LIN {X 0,Y 488.725,Z 711.254,A -85,B 0,C 180,E1 -6470.898,E2 -6470.898} C_VEL
LIN {X 0,Y 488.408,Z 718.913,A -85,B 0,C 180,E1 -6472.143,E2 -6472.143} C_VEL
LIN {X 0,Y 488.185,Z 725.016,A -85,B 0,C 180,E1 -6473.386,E2 -6473.386} C_VEL
LIN {X 0,Y 488.072,Z 729.849,A -85,B 0,C 180,E1 -6474.629,E2 -6474.629} C_VEL
LIN {X 0,Y 488.106,Z 733.551,A -85,B 0,C 180,E1 -6475.871,E2 -6475.871} C_VEL
LIN {X 0,Y 487.981,Z 735.461,A -85,B 0,C 180,E1 -6476.697,E2 -6476.697} C_VEL
LIN {X 0,Y 487.99,Z 736.936,A -85,B 0,C 180,E1 -6477.524,E2 -6477.524} C_VEL
LIN {X 0,Y 487.835,Z 738.611,A -85,B 0,C 180,E1 -6479.174,E2 -6479.174} C_VEL
LIN {X 0,Y 487.82,Z 738.869,A -85,B 0,C 180,E1 -6480,E2 -6480} C_VEL
LIN {X 0,Y 487.835,Z 738.688,A -85,B 0,C 180,E1 -6480.825,E2 -6480.825} C_VEL
LIN {X 0,Y 487.989,Z 737.13,A -85,B 0,C 180,E1 -6482.476,E2 -6482.476} C_VEL
LIN {X 0,Y 487.981,Z 735.745,A -85,B 0,C 180,E1 -6483.302,E2 -6483.302} C_VEL
LIN {X 0,Y 488.067,Z 732.834,A -85,B 0,C 180,E1 -6484.542,E2 -6484.542} C_VEL
LIN {X 0,Y 488.225,Z 727.776,A -85,B 0,C 180,E1 -6486.069,E2 -6486.069} C_VEL
LIN {X 0,Y 488.344,Z 721.731,A -85,B 0,C 180,E1 -6487.442,E2 -6487.442} C_VEL
LIN {X 0,Y 488.606,Z 714.719,A -85,B 0,C 180,E1 -6488.687,E2 -6488.687} C_VEL
LIN {X 0,Y 488.878,Z 705.985,A -85,B 0,C 180,E1 -6489.934,E2 -6489.934} C_VEL
LIN {X 0,Y 489.234,Z 696.973,A -85,B 0,C 180,E1 -6490.973,E2 -6490.973} C_VEL
LIN {X 0,Y 489.603,Z 686.95,A -85,B 0,C 180,E1 -6491.908,E2 -6491.908} C_VEL
LIN {X 0,Y 489.945,Z 676.115,A -85,B 0,C 180,E1 -6492.727,E2 -6492.727} C_VEL
LIN {X 0,Y 490.19,Z 664.496,A -85,B 0,C 180,E1 -6493.42,E2 -6493.42} C_VEL
LIN {X 0,Y 490.575,Z 651.519,A -85,B 0,C 180,E1 -6493.99,E2 -6493.99} C_VEL
LIN {X 0,Y 490.841,Z 638.811,A -85,B 0,C 180,E1 -6494.379,E2 -6494.379} C_VEL
LIN {X 0,Y 491.087,Z 617.625,A -85,B 0,C 180,E1 -6494.742,E2 -6494.742} C_VEL
LIN {X 0,Y 491.674,Z 537.749,A -85,B 0,C 180,E1 -6496.029,E2 -6496.029} C_VEL
LIN {X 0,Y 489.935,Z 527.319,A -85,B 0,C 180,E1 -6496.278,E2 -6496.278} C_VEL
LIN {X 0,Y 490.381,Z 507.251,A -85,B 0,C 180,E1 -6499.246,E2 -6499.246} C_VEL
LIN {X 0,Y 490.847,Z 487.873,A -85,B 0,C 180,E1 -6502.077,E2 -6502.077} C_VEL
LIN {X 0,Y 490.974,Z 472.353,A -85,B 0,C 180,E1 -6504.301,E2 -6504.301} C_VEL
LIN {X 0,Y 488.784,Z 461.229,A -85,B 0,C 180,E1 -6506.011,E2 -6506.011} C_VEL
LIN {X 0,Y 488.728,Z 461.234,A -85,B 0,C 180,E1 -6509.27,E2 -6509.27} C_VEL
LIN {X 0,Y 488.708,Z 461.238,A -85,B 0,C 180,E1 -6512.147,E2 -6512.147} C_VEL
LIN {X 0,Y 488.728,Z 461.23,A -85,B 0,C 180,E1 -6515.114,E2 -6515.114} C_VEL
LIN {X 0,Y 488.685,Z 461.239,A -85,B 0,C 180,E1 -6518.2,E2 -6518.2} C_VEL
LIN {X 0,Y 488.723,Z 461.233,A -85,B 0,C 180,E1 -6520.344,E2 -6520.344} C_VEL
LIN {X 0,Y 488.688,Z 461.238,A -85,B 0,C 180,E1 -6523.654,E2 -6523.654} C_VEL
LIN {X 0,Y 488.689,Z 461.236,A -85,B 0,C 180,E1 -6526.345,E2 -6526.345} C_VEL
LIN {X 0,Y 488.737,Z 461.233,A -85,B 0,C 180,E1 -6529.676,E2 -6529.676} C_VEL
LIN {X 0,Y 488.683,Z 461.234,A -85,B 0,C 180,E1 -6532.841,E2 -6532.841} C_VEL
LIN {X 0,Y 488.735,Z 461.233,A -85,B 0,C 180,E1 -6535.887,E2 -6535.887} C_VEL
LIN {X 0,Y 488.696,Z 461.236,A -85,B 0,C 180,E1 -6538.82,E2 -6538.82} C_VEL
LIN {X 0,Y 488.771,Z 461.307,A -85,B 0,C 180,E1 -6542.154,E2 -6542.154} C_VEL
LIN {X 0,Y 492.591,Z 477.034,A -85,B 0,C 180,E1 -6544.507,E2 -6544.507} C_VEL
LIN {X 0,Y 492.585,Z 483.249,A -85,B 0,C 180,E1 -6545.333,E2 -6545.333} C_VEL
LIN {X 0,Y 491.403,Z 507.9,A -85,B 0,C 180,E1 -6548.515,E2 -6548.515} C_VEL
LIN {X 0,Y 490.794,Z 523.179,A -85,B 0,C 180,E1 -6550.474,E2 -6550.474} C_VEL
LIN {X 0,Y 493.097,Z 539.069,A -85,B 0,C 180,E1 -6550.81,E2 -6550.81} C_VEL
LIN {X 0,Y 491.916,Z 660.89,A -85,B 0,C 180,E1 -6552.701,E2 -6552.701} C_VEL
LIN {X 0,Y 491.605,Z 675.258,A -85,B 0,C 180,E1 -6553.091,E2 -6553.091} C_VEL
LIN {X 0,Y 491.241,Z 688.698,A -85,B 0,C 180,E1 -6553.617,E2 -6553.617} C_VEL
LIN {X 0,Y 490.769,Z 702.208,A -85,B 0,C 180,E1 -6554.317,E2 -6554.317} C_VEL
LIN {X 0,Y 490.228,Z 714.884,A -85,B 0,C 180,E1 -6555.151,E2 -6555.151} C_VEL
LIN {X 0,Y 489.715,Z 726.469,A -85,B 0,C 180,E1 -6556.09,E2 -6556.09} C_VEL
LIN {X 0,Y 489.278,Z 737.113,A -85,B 0,C 180,E1 -6557.135,E2 -6557.135} C_VEL
LIN {X 0,Y 488.939,Z 747.693,A -85,B 0,C 180,E1 -6558.39,E2 -6558.39} C_VEL
LIN {X 0,Y 488.572,Z 756.397,A -85,B 0,C 180,E1 -6559.64,E2 -6559.64} C_VEL
LIN {X 0,Y 488.293,Z 764.689,A -85,B 0,C 180,E1 -6561.098,E2 -6561.098} C_VEL
LIN {X 0,Y 488.084,Z 771.358,A -85,B 0,C 180,E1 -6562.553,E2 -6562.553} C_VEL
LIN {X 0,Y 488.006,Z 776.018,A -85,B 0,C 180,E1 -6563.81,E2 -6563.81} C_VEL
LIN {X 0,Y 487.962,Z 779.592,A -85,B 0,C 180,E1 -6565.041,E2 -6565.041} C_VEL
LIN {X 0,Y 487.959,Z 783.12,A -85,B 0,C 180,E1 -6566.696,E2 -6566.696} C_VEL
LIN {X 0,Y 487.985,Z 784.341,A -85,B 0,C 180,E1 -6567.523,E2 -6567.523} C_VEL
LIN {X 0,Y 487.831,Z 785.722,A -85,B 0,C 180,E1 -6569.173,E2 -6569.173} C_VEL
LIN {X 0,Y 487.83,Z 785.724,A -85,B 0,C 180,E1 -6570.824,E2 -6570.824} C_VEL
LIN {X 0,Y 487.985,Z 784.348,A -85,B 0,C 180,E1 -6572.475,E2 -6572.475} C_VEL
LIN {X 0,Y 487.935,Z 781.551,A -85,B 0,C 180,E1 -6574.129,E2 -6574.129} C_VEL
LIN {X 0,Y 488.022,Z 777.273,A -85,B 0,C 180,E1 -6575.784,E2 -6575.784} C_VEL
LIN {X 0,Y 488.082,Z 771.371,A -85,B 0,C 180,E1 -6577.445,E2 -6577.445} C_VEL
LIN {X 0,Y 488.288,Z 764.706,A -85,B 0,C 180,E1 -6578.9,E2 -6578.9} C_VEL
LIN {X 0,Y 488.577,Z 756.411,A -85,B 0,C 180,E1 -6580.357,E2 -6580.357} C_VEL
LIN {X 0,Y 488.942,Z 747.71,A -85,B 0,C 180,E1 -6581.608,E2 -6581.608} C_VEL
LIN {X 0,Y 489.302,Z 737.14,A -85,B 0,C 180,E1 -6582.862,E2 -6582.862} C_VEL
LIN {X 0,Y 489.779,Z 725.303,A -85,B 0,C 180,E1 -6584.012,E2 -6584.012} C_VEL
LIN {X 0,Y 490.304,Z 713.471,A -85,B 0,C 180,E1 -6584.951,E2 -6584.951} C_VEL
LIN {X 0,Y 490.815,Z 700.451,A -85,B 0,C 180,E1 -6585.786,E2 -6585.786} C_VEL
LIN {X 0,Y 491.313,Z 686.044,A -85,B 0,C 180,E1 -6586.503,E2 -6586.503} C_VEL
LIN {X 0,Y 491.653,Z 672.054,A -85,B 0,C 180,E1 -6587.012,E2 -6587.012} C_VEL
LIN {X 0,Y 491.999,Z 658.343,A -85,B 0,C 180,E1 -6587.348,E2 -6587.348} C_VEL
LIN {X 0,Y 493.037,Z 537.881,A -85,B 0,C 180,E1 -6589.211,E2 -6589.211} C_VEL
LIN {X 0,Y 490.784,Z 522.893,A -85,B 0,C 180,E1 -6589.547,E2 -6589.547} C_VEL
LIN {X 0,Y 491.888,Z 496.801,A -85,B 0,C 180,E1 -6592.912,E2 -6592.912} C_VEL
LIN {X 0,Y 492.731,Z 478.183,A -85,B 0,C 180,E1 -6595.333,E2 -6595.333} C_VEL
LIN {X 0,Y 489.178,Z 462.917,A -85,B 0,C 180,E1 -6597.601,E2 -6597.601} C_VEL
LIN {X 0,Y 488.747,Z 461.229,A -85,B 0,C 180,E1 -6597.86,E2 -6597.86} C_VEL
LIN {X 0,Y 488.715,Z 461.232,A -85,B 0,C 180,E1 -6600.364,E2 -6600.364} C_VEL
LIN {X 0,Y 488.731,Z 461.229,A -85,B 0,C 180,E1 -6603.483,E2 -6603.483} C_VEL
LIN {X 0,Y 488.684,Z 461.233,A -85,B 0,C 180,E1 -6606.355,E2 -6606.355} C_VEL
LIN {X 0,Y 488.743,Z 461.229,A -85,B 0,C 180,E1 -6609.248,E2 -6609.248} C_VEL
LIN {X 0,Y 488.727,Z 461.234,A -85,B 0,C 180,E1 -6612.52,E2 -6612.52} C_VEL
LIN {X 0,Y 488.704,Z 461.232,A -85,B 0,C 180,E1 -6615.198,E2 -6615.198} C_VEL
LIN {X 0,Y 488.727,Z 461.226,A -85,B 0,C 180,E1 -6617.478,E2 -6617.478} C_VEL
LIN {X 0,Y 488.74,Z 461.231,A -85,B 0,C 180,E1 -6620.75,E2 -6620.75} C_VEL
LIN {X 0,Y 488.676,Z 461.226,A -85,B 0,C 180,E1 -6623.868,E2 -6623.868} C_VEL
LIN {X 0,Y 488.73,Z 461.232,A -85,B 0,C 180,E1 -6626.877,E2 -6626.877} C_VEL
LIN {X 0,Y 488.724,Z 461.227,A -85,B 0,C 180,E1 -6629.781,E2 -6629.781} C_VEL
LIN {X 0,Y 488.788,Z 461.223,A -85,B 0,C 180,E1 -6633.054,E2 -6633.054} C_VEL
LIN {X 0,Y 488.683,Z 461.234,A -85,B 0,C 180,E1 -6636.254,E2 -6636.254} C_VEL
LIN {X 0,Y 488.735,Z 461.223,A -85,B 0,C 180,E1 -6639.175,E2 -6639.175} C_VEL
LIN {X 0,Y 488.748,Z 461.225,A -85,B 0,C 180,E1 -6641.627,E2 -6641.627} C_VEL
LIN {X 0,Y 488.75,Z 461.228,A -85,B 0,C 180,E1 -6644.999,E2 -6644.999} C_VEL
LIN {X 0,Y 488.822,Z 461.22,A -85,B 0,C 180,E1 -6648.388,E2 -6648.388} C_VEL
LIN {X 0,Y 488.807,Z 461.218,A -85,B 0,C 180,E1 -6651.734,E2 -6651.734} C_VEL
LIN {X 0,Y 488.852,Z 461.211,A -85,B 0,C 180,E1 -6654.224,E2 -6654.224} C_VEL
LIN {X 0,Y 488.952,Z 461.198,A -85,B 0,C 180,E1 -6657.529,E2 -6657.529} C_VEL
LIN {X 0,Y 488.958,Z 461.199,A -85,B 0,C 180,E1 -6660,E2 -6660} C_VEL
LIN {X 0,Y 488.951,Z 461.205,A -85,B 0,C 180,E1 -6662.472,E2 -6662.472} C_VEL
LIN {X 0,Y 488.845,Z 461.213,A -85,B 0,C 180,E1 -6665.776,E2 -6665.776} C_VEL
LIN {X 0,Y 488.808,Z 461.22,A -85,B 0,C 180,E1 -6668.267,E2 -6668.267} C_VEL
LIN {X 0,Y 488.819,Z 461.216,A -85,B 0,C 180,E1 -6671.612,E2 -6671.612} C_VEL
LIN {X 0,Y 488.754,Z 461.227,A -85,B 0,C 180,E1 -6675.001,E2 -6675.001} C_VEL
LIN {X 0,Y 488.744,Z 461.229,A -85,B 0,C 180,E1 -6678.443,E2 -6678.443} C_VEL
LIN {X 0,Y 488.697,Z 461.232,A -85,B 0,C 180,E1 -6681.071,E2 -6681.071} C_VEL
LIN {X 0,Y 488.684,Z 461.233,A -85,B 0,C 180,E1 -6683.746,E2 -6683.746} C_VEL
LIN {X 0,Y 488.789,Z 461.222,A -85,B 0,C 180,E1 -6686.946,E2 -6686.946} C_VEL
LIN {X 0,Y 488.71,Z 461.234,A -85,B 0,C 180,E1 -6690.366,E2 -6690.366} C_VEL
LIN {X 0,Y 488.728,Z 461.226,A -85,B 0,C 180,E1 -6693.486,E2 -6693.486} C_VEL
LIN {X 0,Y 488.682,Z 461.241,A -85,B 0,C 180,E1 -6696.357,E2 -6696.357} C_VEL
LIN {X 0,Y 488.741,Z 461.227,A -85,B 0,C 180,E1 -6699.251,E2 -6699.251} C_VEL
LIN {X 0,Y 488.684,Z 461.24,A -85,B 0,C 180,E1 -6702.527,E2 -6702.527} C_VEL
LIN {X 0,Y 488.706,Z 461.231,A -85,B 0,C 180,E1 -6705.2,E2 -6705.2} C_VEL
LIN {X 0,Y 488.73,Z 461.228,A -85,B 0,C 180,E1 -6707.481,E2 -6707.481} C_VEL
LIN {X 0,Y 488.745,Z 461.231,A -85,B 0,C 180,E1 -6710.752,E2 -6710.752} C_VEL
LIN {X 0,Y 488.682,Z 461.233,A -85,B 0,C 180,E1 -6713.87,E2 -6713.87} C_VEL
LIN {X 0,Y 488.736,Z 461.232,A -85,B 0,C 180,E1 -6716.879,E2 -6716.879} C_VEL
LIN {X 0,Y 488.732,Z 461.231,A -85,B 0,C 180,E1 -6719.783,E2 -6719.783} C_VEL
LIN {X 0,Y 488.792,Z 461.226,A -85,B 0,C 180,E1 -6723.11,E2 -6723.11} C_VEL
LIN {X 0,Y 488.533,Z 461.627,A -85,B 0,C 180,E1 -6723.564,E2 -6723.564} C_VEL
LIN {X 0,Y 487.572,Z 463.402,A -85,B 0,C 180,E1 -6724.212,E2 -6724.212} C_VEL
LIN {X 0,Y 486.316,Z 466.116,A -85,B 0,C 180,E1 -6724.816,E2 -6724.816} C_VEL
LIN {X 0,Y 484.792,Z 470.694,A -85,B 0,C 180,E1 -6725.6,E2 -6725.6} C_VEL
LIN {X 0,Y 484.379,Z 475.251,A -85,B 0,C 180,E1 -6726.389,E2 -6726.389} C_VEL
LIN {X 0,Y 483.995,Z 487.151,A -85,B 0,C 180,E1 -6728.472,E2 -6728.472} C_VEL
LIN {X 0,Y 483.111,Z 507.748,A -85,B 0,C 180,E1 -6731.994,E2 -6731.994} C_VEL
LIN {X 0,Y 482.787,Z 515.697,A -85,B 0,C 180,E1 -6733.327,E2 -6733.327} C_VEL
LIN {X 0,Y 485.47,Z 530.483,A -85,B 0,C 180,E1 -6733.646,E2 -6733.646} C_VEL
LIN {X 0,Y 485.028,Z 626.011,A -85,B 0,C 180,E1 -6734.99,E2 -6734.99} C_VEL
LIN {X 0,Y 484.776,Z 638.769,A -85,B 0,C 180,E1 -6735.331,E2 -6735.331} C_VEL
LIN {X 0,Y 484.401,Z 651.155,A -85,B 0,C 180,E1 -6735.829,E2 -6735.829} C_VEL
LIN {X 0,Y 484.02,Z 662.666,A -85,B 0,C 180,E1 -6736.461,E2 -6736.461} C_VEL
LIN {X 0,Y 483.555,Z 673.193,A -85,B 0,C 180,E1 -6737.201,E2 -6737.201} C_VEL
LIN {X 0,Y 483.049,Z 683.796,A -85,B 0,C 180,E1 -6738.142,E2 -6738.142} C_VEL
LIN {X 0,Y 482.618,Z 692.492,A -85,B 0,C 180,E1 -6739.089,E2 -6739.089} C_VEL
LIN {X 0,Y 482.109,Z 701.921,A -85,B 0,C 180,E1 -6740.35,E2 -6740.35} C_VEL
LIN {X 0,Y 481.674,Z 709.481,A -85,B 0,C 180,E1 -6741.611,E2 -6741.611} C_VEL
LIN {X 0,Y 481.359,Z 715.713,A -85,B 0,C 180,E1 -6742.914,E2 -6742.914} C_VEL
LIN {X 0,Y 481.15,Z 720.373,A -85,B 0,C 180,E1 -6744.133,E2 -6744.133} C_VEL
LIN {X 0,Y 481.041,Z 724.131,A -85,B 0,C 180,E1 -6745.392,E2 -6745.392} C_VEL
LIN {X 0,Y 480.984,Z 726.915,A -85,B 0,C 180,E1 -6746.65,E2 -6746.65} C_VEL
LIN {X 0,Y 480.939,Z 728.241,A -85,B 0,C 180,E1 -6747.489,E2 -6747.489} C_VEL
LIN {X 0,Y 480.762,Z 729.781,A -85,B 0,C 180,E1 -6749.163,E2 -6749.163} C_VEL
LIN {X 0,Y 480.748,Z 730.004,A -85,B 0,C 180,E1 -6750.001,E2 -6750.001} C_VEL
LIN {X 0,Y 480.826,Z 729.271,A -85,B 0,C 180,E1 -6751.676,E2 -6751.676} C_VEL
LIN {X 0,Y 480.937,Z 728.348,A -85,B 0,C 180,E1 -6752.514,E2 -6752.514} C_VEL
LIN {X 0,Y 480.961,Z 727.06,A -85,B 0,C 180,E1 -6753.352,E2 -6753.352} C_VEL
LIN {X 0,Y 481.034,Z 724.342,A -85,B 0,C 180,E1 -6754.61,E2 -6754.61} C_VEL
LIN {X 0,Y 481.147,Z 720.657,A -85,B 0,C 180,E1 -6755.87,E2 -6755.87} C_VEL
LIN {X 0,Y 481.397,Z 715.111,A -85,B 0,C 180,E1 -6757.319,E2 -6757.319} C_VEL
LIN {X 0,Y 481.726,Z 708.806,A -85,B 0,C 180,E1 -6758.601,E2 -6758.601} C_VEL
LIN {X 0,Y 482.108,Z 701.082,A -85,B 0,C 180,E1 -6759.864,E2 -6759.864} C_VEL
LIN {X 0,Y 482.615,Z 691.481,A -85,B 0,C 180,E1 -6761.126,E2 -6761.126} C_VEL
LIN {X 0,Y 483.177,Z 681.429,A -85,B 0,C 180,E1 -6762.177,E2 -6762.177} C_VEL
LIN {X 0,Y 483.684,Z 670.239,A -85,B 0,C 180,E1 -6763.111,E2 -6763.111} C_VEL
LIN {X 0,Y 484.171,Z 658.857,A -85,B 0,C 180,E1 -6763.858,E2 -6763.858} C_VEL
LIN {X 0,Y 484.577,Z 647.318,A -85,B 0,C 180,E1 -6764.436,E2 -6764.436} C_VEL
LIN {X 0,Y 484.864,Z 634.808,A -85,B 0,C 180,E1 -6764.883,E2 -6764.883} C_VEL
LIN {X 0,Y 485.089,Z 621.87,A -85,B 0,C 180,E1 -6765.171,E2 -6765.171} C_VEL
LIN {X 0,Y 485.331,Z 529.087,A -85,B 0,C 180,E1 -6766.469,E2 -6766.469} C_VEL
LIN {X 0,Y 482.801,Z 515.558,A -85,B 0,C 180,E1 -6766.786,E2 -6766.786} C_VEL
LIN {X 0,Y 483.399,Z 499.245,A -85,B 0,C 180,E1 -6769.536,E2 -6769.536} C_VEL
LIN {X 0,Y 484.17,Z 482.676,A -85,B 0,C 180,E1 -6772.399,E2 -6772.399} C_VEL
LIN {X 0,Y 484.393,Z 475.065,A -85,B 0,C 180,E1 -6773.734,E2 -6773.734} C_VEL
LIN {X 0,Y 481.723,Z 462.108,A -85,B 0,C 180,E1 -6776.248,E2 -6776.248} C_VEL
LIN {X 0,Y 481.684,Z 462.113,A -85,B 0,C 180,E1 -6778.904,E2 -6778.904} C_VEL
LIN {X 0,Y 481.663,Z 462.113,A -85,B 0,C 180,E1 -6782.19,E2 -6782.19} C_VEL
LIN {X 0,Y 481.694,Z 462.105,A -85,B 0,C 180,E1 -6784.683,E2 -6784.683} C_VEL
LIN {X 0,Y 481.661,Z 462.111,A -85,B 0,C 180,E1 -6788.008,E2 -6788.008} C_VEL
LIN {X 0,Y 481.669,Z 462.108,A -85,B 0,C 180,E1 -6791.041,E2 -6791.041} C_VEL
LIN {X 0,Y 481.665,Z 462.106,A -85,B 0,C 180,E1 -6794.36,E2 -6794.36} C_VEL
LIN {X 0,Y 481.649,Z 462.11,A -85,B 0,C 180,E1 -6796.852,E2 -6796.852} C_VEL
LIN {X 0,Y 481.683,Z 462.108,A -85,B 0,C 180,E1 -6800.06,E2 -6800.06} C_VEL
LIN {X 0,Y 481.635,Z 462.111,A -85,B 0,C 180,E1 -6803.254,E2 -6803.254} C_VEL
LIN {X 0,Y 481.716,Z 462.103,A -85,B 0,C 180,E1 -6806.33,E2 -6806.33} C_VEL
LIN {X 0,Y 481.657,Z 462.114,A -85,B 0,C 180,E1 -6809.417,E2 -6809.417} C_VEL
LIN {X 0,Y 481.706,Z 462.107,A -85,B 0,C 180,E1 -6812.168,E2 -6812.168} C_VEL
LIN {X 0,Y 481.761,Z 462.29,A -85,B 0,C 180,E1 -6813.61,E2 -6813.61} C_VEL
LIN {X 0,Y 484.205,Z 474.142,A -85,B 0,C 180,E1 -6815.565,E2 -6815.565} C_VEL
LIN {X 0,Y 484.167,Z 483.006,A -85,B 0,C 180,E1 -6816.926,E2 -6816.926} C_VEL
LIN {X 0,Y 483.541,Z 503.362,A -85,B 0,C 180,E1 -6820.028,E2 -6820.028} C_VEL
LIN {X 0,Y 482.967,Z 523.364,A -85,B 0,C 180,E1 -6823.08,E2 -6823.08} C_VEL
LIN {X 0,Y 482.888,Z 526.537,A -85,B 0,C 180,E1 -6823.562,E2 -6823.562} C_VEL
LIN {X 0,Y 484.92,Z 539.144,A -85,B 0,C 180,E1 -6823.859,E2 -6823.859} C_VEL
LIN {X 0,Y 483.987,Z 636.668,A -85,B 0,C 180,E1 -6825.44,E2 -6825.44} C_VEL
LIN {X 0,Y 483.758,Z 649.432,A -85,B 0,C 180,E1 -6825.809,E2 -6825.809} C_VEL
LIN {X 0,Y 483.415,Z 661.772,A -85,B 0,C 180,E1 -6826.335,E2 -6826.335} C_VEL
LIN {X 0,Y 483.085,Z 673.368,A -85,B 0,C 180,E1 -6826.993,E2 -6826.993} C_VEL
LIN {X 0,Y 482.756,Z 684.635,A -85,B 0,C 180,E1 -6827.813,E2 -6827.813} C_VEL
LIN {X 0,Y 482.283,Z 696.06,A -85,B 0,C 180,E1 -6828.867,E2 -6828.867} C_VEL
LIN {X 0,Y 481.923,Z 705.281,A -85,B 0,C 180,E1 -6829.921,E2 -6829.921} C_VEL
LIN {X 0,Y 481.586,Z 714.167,A -85,B 0,C 180,E1 -6831.186,E2 -6831.186} C_VEL
LIN {X 0,Y 481.289,Z 721.327,A -85,B 0,C 180,E1 -6832.448,E2 -6832.448} C_VEL
LIN {X 0,Y 481.135,Z 726.739,A -85,B 0,C 180,E1 -6833.637,E2 -6833.637} C_VEL
LIN {X 0,Y 480.915,Z 731.506,A -85,B 0,C 180,E1 -6834.97,E2 -6834.97} C_VEL
LIN {X 0,Y 481.021,Z 733.841,A -85,B 0,C 180,E1 -6835.811,E2 -6835.811} C_VEL
LIN {X 0,Y 480.913,Z 735.764,A -85,B 0,C 180,E1 -6836.649,E2 -6836.649} C_VEL
LIN {X 0,Y 480.897,Z 737.251,A -85,B 0,C 180,E1 -6837.487,E2 -6837.487} C_VEL
LIN {X 0,Y 480.761,Z 738.938,A -85,B 0,C 180,E1 -6839.162,E2 -6839.162} C_VEL
LIN {X 0,Y 480.744,Z 739.2,A -85,B 0,C 180,E1 -6840,E2 -6840} C_VEL
LIN {X 0,Y 480.761,Z 739.019,A -85,B 0,C 180,E1 -6840.837,E2 -6840.837} C_VEL
LIN {X 0,Y 480.911,Z 737.457,A -85,B 0,C 180,E1 -6842.513,E2 -6842.513} C_VEL
LIN {X 0,Y 480.913,Z 736.064,A -85,B 0,C 180,E1 -6843.351,E2 -6843.351} C_VEL
LIN {X 0,Y 480.982,Z 733.14,A -85,B 0,C 180,E1 -6844.609,E2 -6844.609} C_VEL
LIN {X 0,Y 481.134,Z 729.148,A -85,B 0,C 180,E1 -6845.869,E2 -6845.869} C_VEL
LIN {X 0,Y 481.209,Z 723.972,A -85,B 0,C 180,E1 -6847.131,E2 -6847.131} C_VEL
LIN {X 0,Y 481.49,Z 717.445,A -85,B 0,C 180,E1 -6848.393,E2 -6848.393} C_VEL
LIN {X 0,Y 481.738,Z 709.334,A -85,B 0,C 180,E1 -6849.658,E2 -6849.658} C_VEL
LIN {X 0,Y 482.079,Z 700.952,A -85,B 0,C 180,E1 -6850.712,E2 -6850.712} C_VEL
LIN {X 0,Y 482.522,Z 690.632,A -85,B 0,C 180,E1 -6851.766,E2 -6851.766} C_VEL
LIN {X 0,Y 482.886,Z 680.426,A -85,B 0,C 180,E1 -6852.61,E2 -6852.61} C_VEL
LIN {X 0,Y 483.182,Z 668.326,A -85,B 0,C 180,E1 -6853.399,E2 -6853.399} C_VEL
LIN {X 0,Y 483.583,Z 655.358,A -85,B 0,C 180,E1 -6854.035,E2 -6854.035} C_VEL
LIN {X 0,Y 483.889,Z 642.229,A -85,B 0,C 180,E1 -6854.482,E2 -6854.482} C_VEL
LIN {X 0,Y 484.068,Z 628.396,A -85,B 0,C 180,E1 -6854.773,E2 -6854.773} C_VEL
LIN {X 0,Y 484.879,Z 538.539,A -85,B 0,C 180,E1 -6856.253,E2 -6856.253} C_VEL
LIN {X 0,Y 483.066,Z 527.717,A -85,B 0,C 180,E1 -6856.527,E2 -6856.527} C_VEL
LIN {X 0,Y 483.499,Z 507.474,A -85,B 0,C 180,E1 -6859.531,E2 -6859.531} C_VEL
LIN {X 0,Y 483.941,Z 490.703,A -85,B 0,C 180,E1 -6862.003,E2 -6862.003} C_VEL
LIN {X 0,Y 484.299,Z 475.446,A -85,B 0,C 180,E1 -6864.202,E2 -6864.202} C_VEL
LIN {X 0,Y 482.705,Z 466.129,A -85,B 0,C 180,E1 -6865.626,E2 -6865.626} C_VEL
LIN {X 0,Y 481.73,Z 462.107,A -85,B 0,C 180,E1 -6866.275,E2 -6866.275} C_VEL
LIN {X 0,Y 481.683,Z 462.112,A -85,B 0,C 180,E1 -6868.903,E2 -6868.903} C_VEL
LIN {X 0,Y 481.662,Z 462.116,A -85,B 0,C 180,E1 -6872.189,E2 -6872.189} C_VEL
LIN {X 0,Y 481.698,Z 462.108,A -85,B 0,C 180,E1 -6874.681,E2 -6874.681} C_VEL
LIN {X 0,Y 481.66,Z 462.116,A -85,B 0,C 180,E1 -6878.007,E2 -6878.007} C_VEL
LIN {X 0,Y 481.661,Z 462.11,A -85,B 0,C 180,E1 -6881.041,E2 -6881.041} C_VEL
LIN {X 0,Y 481.659,Z 462.112,A -85,B 0,C 180,E1 -6884.457,E2 -6884.457} C_VEL
LIN {X 0,Y 481.652,Z 462.116,A -85,B 0,C 180,E1 -6887.839,E2 -6887.839} C_VEL
LIN {X 0,Y 481.665,Z 462.107,A -85,B 0,C 180,E1 -6890.653,E2 -6890.653} C_VEL
LIN {X 0,Y 481.632,Z 462.118,A -85,B 0,C 180,E1 -6893.376,E2 -6893.376} C_VEL
LIN {X 0,Y 481.714,Z 462.105,A -85,B 0,C 180,E1 -6896.329,E2 -6896.329} C_VEL
LIN {X 0,Y 481.655,Z 462.117,A -85,B 0,C 180,E1 -6899.417,E2 -6899.417} C_VEL
LIN {X 0,Y 481.709,Z 462.126,A -85,B 0,C 180,E1 -6901.842,E2 -6901.842} C_VEL
LIN {X 0,Y 485.587,Z 477.99,A -85,B 0,C 180,E1 -6904.265,E2 -6904.265} C_VEL
LIN {X 0,Y 485.926,Z 481.392,A -85,B 0,C 180,E1 -6904.743,E2 -6904.743} C_VEL
LIN {X 0,Y 484.664,Z 505.062,A -85,B 0,C 180,E1 -6907.85,E2 -6907.85} C_VEL
LIN {X 0,Y 483.87,Z 522.955,A -85,B 0,C 180,E1 -6910.197,E2 -6910.197} C_VEL
LIN {X 0,Y 486.32,Z 539.434,A -85,B 0,C 180,E1 -6910.563,E2 -6910.563} C_VEL
LIN {X 0,Y 485.078,Z 660.109,A -85,B 0,C 180,E1 -6912.476,E2 -6912.476} C_VEL
LIN {X 0,Y 484.722,Z 674.54,A -85,B 0,C 180,E1 -6912.871,E2 -6912.871} C_VEL
LIN {X 0,Y 484.35,Z 688.164,A -85,B 0,C 180,E1 -6913.41,E2 -6913.41} C_VEL
LIN {X 0,Y 483.851,Z 701.149,A -85,B 0,C 180,E1 -6914.087,E2 -6914.087} C_VEL
LIN {X 0,Y 483.294,Z 713.953,A -85,B 0,C 180,E1 -6914.933,E2 -6914.933} C_VEL
LIN {X 0,Y 482.774,Z 725.639,A -85,B 0,C 180,E1 -6915.886,E2 -6915.886} C_VEL
LIN {X 0,Y 482.279,Z 736.362,A -85,B 0,C 180,E1 -6916.945,E2 -6916.945} C_VEL
LIN {X 0,Y 481.917,Z 747.023,A -85,B 0,C 180,E1 -6918.218,E2 -6918.218} C_VEL
LIN {X 0,Y 481.529,Z 755.788,A -85,B 0,C 180,E1 -6919.487,E2 -6919.487} C_VEL
LIN {X 0,Y 481.225,Z 764.136,A -85,B 0,C 180,E1 -6920.966,E2 -6920.966} C_VEL
LIN {X 0,Y 481.009,Z 770.847,A -85,B 0,C 180,E1 -6922.443,E2 -6922.443} C_VEL
LIN {X 0,Y 480.909,Z 775.917,A -85,B 0,C 180,E1 -6923.841,E2 -6923.841} C_VEL
LIN {X 0,Y 480.896,Z 779.136,A -85,B 0,C 180,E1 -6924.968,E2 -6924.968} C_VEL
LIN {X 0,Y 480.884,Z 782.69,A -85,B 0,C 180,E1 -6926.648,E2 -6926.648} C_VEL
LIN {X 0,Y 480.822,Z 784.791,A -85,B 0,C 180,E1 -6928.324,E2 -6928.324} C_VEL
LIN {X 0,Y 480.741,Z 785.487,A -85,B 0,C 180,E1 -6929.999,E2 -6929.999} C_VEL
LIN {X 0,Y 480.822,Z 784.795,A -85,B 0,C 180,E1 -6931.674,E2 -6931.674} C_VEL
LIN {X 0,Y 480.883,Z 782.7,A -85,B 0,C 180,E1 -6933.35,E2 -6933.35} C_VEL
LIN {X 0,Y 480.896,Z 779.152,A -85,B 0,C 180,E1 -6935.029,E2 -6935.029} C_VEL
LIN {X 0,Y 480.961,Z 774.047,A -85,B 0,C 180,E1 -6936.712,E2 -6936.712} C_VEL
LIN {X 0,Y 481.08,Z 769.096,A -85,B 0,C 180,E1 -6937.976,E2 -6937.976} C_VEL
LIN {X 0,Y 481.332,Z 761.936,A -85,B 0,C 180,E1 -6939.453,E2 -6939.453} C_VEL
LIN {X 0,Y 481.657,Z 753.03,A -85,B 0,C 180,E1 -6940.933,E2 -6940.933} C_VEL
LIN {X 0,Y 481.908,Z 744.117,A -85,B 0,C 180,E1 -6942.153,E2 -6942.153} C_VEL
LIN {X 0,Y 482.459,Z 733.391,A -85,B 0,C 180,E1 -6943.37,E2 -6943.37} C_VEL
LIN {X 0,Y 482.962,Z 722.068,A -85,B 0,C 180,E1 -6944.429,E2 -6944.429} C_VEL
LIN {X 0,Y 483.529,Z 709.56,A -85,B 0,C 180,E1 -6945.381,E2 -6945.381} C_VEL
LIN {X 0,Y 483.983,Z 696.444,A -85,B 0,C 180,E1 -6946.18,E2 -6946.18} C_VEL
LIN {X 0,Y 484.433,Z 683.35,A -85,B 0,C 180,E1 -6946.801,E2 -6946.801} C_VEL
LIN {X 0,Y 484.864,Z 669.495,A -85,B 0,C 180,E1 -6947.285,E2 -6947.285} C_VEL
LIN {X 0,Y 485.2,Z 654.571,A -85,B 0,C 180,E1 -6947.626,E2 -6947.626} C_VEL
LIN {X 0,Y 486.307,Z 539.649,A -85,B 0,C 180,E1 -6949.432,E2 -6949.432} C_VEL
LIN {X 0,Y 483.91,Z 522.826,A -85,B 0,C 180,E1 -6949.813,E2 -6949.813} C_VEL
LIN {X 0,Y 485.006,Z 498.304,A -85,B 0,C 180,E1 -6953.031,E2 -6953.031} C_VEL
LIN {X 0,Y 485.887,Z 479.709,A -85,B 0,C 180,E1 -6955.486,E2 -6955.486} C_VEL
LIN {X 0,Y 482.247,Z 464.453,A -85,B 0,C 180,E1 -6957.796,E2 -6957.796} C_VEL
LIN {X 0,Y 481.716,Z 462.105,A -85,B 0,C 180,E1 -6958.184,E2 -6958.184} C_VEL
LIN {X 0,Y 481.649,Z 462.114,A -85,B 0,C 180,E1 -6960.709,E2 -6960.709} C_VEL
LIN {X 0,Y 481.691,Z 462.105,A -85,B 0,C 180,E1 -6963.732,E2 -6963.732} C_VEL
LIN {X 0,Y 481.625,Z 462.118,A -85,B 0,C 180,E1 -6966.745,E2 -6966.745} C_VEL
LIN {X 0,Y 481.687,Z 462.107,A -85,B 0,C 180,E1 -6969.938,E2 -6969.938} C_VEL
LIN {X 0,Y 481.677,Z 462.108,A -85,B 0,C 180,E1 -6973.294,E2 -6973.294} C_VEL
LIN {X 0,Y 481.681,Z 462.11,A -85,B 0,C 180,E1 -6976.845,E2 -6976.845} C_VEL
LIN {X 0,Y 481.684,Z 462.104,A -85,B 0,C 180,E1 -6980.06,E2 -6980.06} C_VEL
LIN {X 0,Y 481.621,Z 462.105,A -85,B 0,C 180,E1 -6983.253,E2 -6983.253} C_VEL
LIN {X 0,Y 481.699,Z 462.103,A -85,B 0,C 180,E1 -6986.329,E2 -6986.329} C_VEL
LIN {X 0,Y 481.649,Z 462.109,A -85,B 0,C 180,E1 -6989.415,E2 -6989.415} C_VEL
LIN {X 0,Y 481.692,Z 462.105,A -85,B 0,C 180,E1 -6992.168,E2 -6992.168} C_VEL
LIN {X 0,Y 481.708,Z 462.104,A -85,B 0,C 180,E1 -6994.969,E2 -6994.969} C_VEL
LIN {X 0,Y 481.642,Z 462.097,A -85,B 0,C 180,E1 -6997.704,E2 -6997.704} C_VEL
LIN {X 0,Y 481.697,Z 462.103,A -85,B 0,C 180,E1 -7000.393,E2 -7000.393} C_VEL
LIN {X 0,Y 481.681,Z 462.106,A -85,B 0,C 180,E1 -7003.034,E2 -7003.034} C_VEL
LIN {X 0,Y 481.68,Z 462.105,A -85,B 0,C 180,E1 -7005.639,E2 -7005.639} C_VEL
LIN {X 0,Y 481.784,Z 462.095,A -85,B 0,C 180,E1 -7008.216,E2 -7008.216} C_VEL
LIN {X 0,Y 481.753,Z 462.096,A -85,B 0,C 180,E1 -7011.612,E2 -7011.612} C_VEL
LIN {X 0,Y 481.812,Z 462.086,A -85,B 0,C 180,E1 -7014.14,E2 -7014.14} C_VEL
LIN {X 0,Y 481.919,Z 462.074,A -85,B 0,C 180,E1 -7017.493,E2 -7017.493} C_VEL
LIN {X 0,Y 481.929,Z 462.074,A -85,B 0,C 180,E1 -7020,E2 -7020} C_VEL
LIN {X 0,Y 481.918,Z 462.08,A -85,B 0,C 180,E1 -7022.508,E2 -7022.508} C_VEL
LIN {X 0,Y 481.806,Z 462.091,A -85,B 0,C 180,E1 -7025.861,E2 -7025.861} C_VEL
LIN {X 0,Y 481.753,Z 462.099,A -85,B 0,C 180,E1 -7028.389,E2 -7028.389} C_VEL
LIN {X 0,Y 481.784,Z 462.093,A -85,B 0,C 180,E1 -7031.784,E2 -7031.784} C_VEL
LIN {X 0,Y 481.733,Z 462.1,A -85,B 0,C 180,E1 -7035.225,E2 -7035.225} C_VEL
LIN {X 0,Y 481.702,Z 462.109,A -85,B 0,C 180,E1 -7038.722,E2 -7038.722} C_VEL
LIN {X 0,Y 481.637,Z 462.109,A -85,B 0,C 180,E1 -7041.395,E2 -7041.395} C_VEL
LIN {X 0,Y 481.667,Z 462.11,A -85,B 0,C 180,E1 -7044.114,E2 -7044.114} C_VEL
LIN {X 0,Y 481.742,Z 462.098,A -85,B 0,C 180,E1 -7047.141,E2 -7047.141} C_VEL
LIN {X 0,Y 481.679,Z 462.105,A -85,B 0,C 180,E1 -7049.741,E2 -7049.741} C_VEL
LIN {X 0,Y 481.665,Z 462.112,A -85,B 0,C 180,E1 -7052.675,E2 -7052.675} C_VEL
LIN {X 0,Y 481.636,Z 462.112,A -85,B 0,C 180,E1 -7055.71,E2 -7055.71} C_VEL
LIN {X 0,Y 481.712,Z 462.102,A -85,B 0,C 180,E1 -7059.356,E2 -7059.356} C_VEL
LIN {X 0,Y 481.642,Z 462.116,A -85,B 0,C 180,E1 -7062.162,E2 -7062.162} C_VEL
LIN {X 0,Y 481.654,Z 462.109,A -85,B 0,C 180,E1 -7065.544,E2 -7065.544} C_VEL
LIN {X 0,Y 481.668,Z 462.112,A -85,B 0,C 180,E1 -7068.086,E2 -7068.086} C_VEL
LIN {X 0,Y 481.699,Z 462.105,A -85,B 0,C 180,E1 -7071.145,E2 -7071.145} C_VEL
LIN {X 0,Y 481.665,Z 462.112,A -85,B 0,C 180,E1 -7074.796,E2 -7074.796} C_VEL
LIN {X 0,Y 481.671,Z 462.109,A -85,B 0,C 180,E1 -7077.327,E2 -7077.327} C_VEL
LIN {X 0,Y 481.686,Z 462.111,A -85,B 0,C 180,E1 -7080.261,E2 -7080.261} C_VEL
LIN {X 0,Y 481.726,Z 462.106,A -85,B 0,C 180,E1 -7083.58,E2 -7083.58} C_VEL
LIN {X 0,Y 481.754,Z 462.261,A -85,B 0,C 180,E1 -7083.902,E2 -7083.902} C_VEL
LIN {X 0,Y 484.379,Z 475.251,A -85,B 0,C 180,E1 -7086.389,E2 -7086.389} C_VEL
LIN {X 0,Y 483.925,Z 478.596,A -85,B 0,C 180,E1 -7086.958,E2 -7086.958} C_VEL
LIN {X 0,Y 482.338,Z 482.1,A -85,B 0,C 180,E1 -7087.494,E2 -7087.494} C_VEL
LIN {X 0,Y 477.7,Z 490.388,A -85,B 0,C 180,E1 -7088.725,E2 -7088.725} C_VEL
LIN {X 0,Y 476.799,Z 493.87,A -85,B 0,C 180,E1 -7089.297,E2 -7089.297} C_VEL
LIN {X 0,Y 476.06,Z 510.529,A -85,B 0,C 180,E1 -7092.163,E2 -7092.163} C_VEL
LIN {X 0,Y 475.886,Z 515.871,A -85,B 0,C 180,E1 -7093.056,E2 -7093.056} C_VEL
LIN {X 0,Y 478.725,Z 530.777,A -85,B 0,C 180,E1 -7093.387,E2 -7093.387} C_VEL
LIN {X 0,Y 478.249,Z 626.376,A -85,B 0,C 180,E1 -7094.745,E2 -7094.745} C_VEL
LIN {X 0,Y 477.989,Z 639.149,A -85,B 0,C 180,E1 -7095.091,E2 -7095.091} C_VEL
LIN {X 0,Y 477.578,Z 652.109,A -85,B 0,C 180,E1 -7095.622,E2 -7095.622} C_VEL
LIN {X 0,Y 477.17,Z 663.496,A -85,B 0,C 180,E1 -7096.262,E2 -7096.262} C_VEL
LIN {X 0,Y 476.67,Z 675.158,A -85,B 0,C 180,E1 -7097.119,E2 -7097.119} C_VEL
LIN {X 0,Y 476.022,Z 685.515,A -85,B 0,C 180,E1 -7098.072,E2 -7098.072} C_VEL
LIN {X 0,Y 475.569,Z 694.858,A -85,B 0,C 180,E1 -7099.141,E2 -7099.141} C_VEL
LIN {X 0,Y 475.157,Z 702.513,A -85,B 0,C 180,E1 -7100.208,E2 -7100.208} C_VEL
LIN {X 0,Y 474.69,Z 710.027,A -85,B 0,C 180,E1 -7101.487,E2 -7101.487} C_VEL
LIN {X 0,Y 474.328,Z 716.227,A -85,B 0,C 180,E1 -7102.809,E2 -7102.809} C_VEL
LIN {X 0,Y 474.109,Z 720.855,A -85,B 0,C 180,E1 -7104.045,E2 -7104.045} C_VEL
LIN {X 0,Y 473.982,Z 724.587,A -85,B 0,C 180,E1 -7105.323,E2 -7105.323} C_VEL
LIN {X 0,Y 473.912,Z 727.351,A -85,B 0,C 180,E1 -7106.6,E2 -7106.6} C_VEL
LIN {X 0,Y 473.88,Z 728.663,A -85,B 0,C 180,E1 -7107.451,E2 -7107.451} C_VEL
LIN {X 0,Y 473.691,Z 730.192,A -85,B 0,C 180,E1 -7109.151,E2 -7109.151} C_VEL
LIN {X 0,Y 473.674,Z 730.412,A -85,B 0,C 180,E1 -7110.001,E2 -7110.001} C_VEL
LIN {X 0,Y 473.761,Z 729.687,A -85,B 0,C 180,E1 -7111.701,E2 -7111.701} C_VEL
LIN {X 0,Y 473.878,Z 728.771,A -85,B 0,C 180,E1 -7112.551,E2 -7112.551} C_VEL
LIN {X 0,Y 473.995,Z 725.811,A -85,B 0,C 180,E1 -7114.253,E2 -7114.253} C_VEL
LIN {X 0,Y 473.981,Z 722.499,A -85,B 0,C 180,E1 -7115.532,E2 -7115.532} C_VEL
LIN {X 0,Y 474.243,Z 718.065,A -85,B 0,C 180,E1 -7116.829,E2 -7116.829} C_VEL
LIN {X 0,Y 474.587,Z 711.548,A -85,B 0,C 180,E1 -7118.303,E2 -7118.303} C_VEL
LIN {X 0,Y 475.004,Z 704.41,A -85,B 0,C 180,E1 -7119.583,E2 -7119.583} C_VEL
LIN {X 0,Y 475.515,Z 695.557,A -85,B 0,C 180,E1 -7120.863,E2 -7120.863} C_VEL
LIN {X 0,Y 475.994,Z 686.368,A -85,B 0,C 180,E1 -7121.931,E2 -7121.931} C_VEL
LIN {X 0,Y 476.661,Z 675.195,A -85,B 0,C 180,E1 -7122.968,E2 -7122.968} C_VEL
LIN {X 0,Y 477.11,Z 664.793,A -85,B 0,C 180,E1 -7123.742,E2 -7123.742} C_VEL
LIN {X 0,Y 477.637,Z 652.811,A -85,B 0,C 180,E1 -7124.432,E2 -7124.432} C_VEL
LIN {X 0,Y 477.952,Z 640.12,A -85,B 0,C 180,E1 -7124.967,E2 -7124.967} C_VEL
LIN {X 0,Y 478.273,Z 626.654,A -85,B 0,C 180,E1 -7125.338,E2 -7125.338} C_VEL
LIN {X 0,Y 478.743,Z 531.309,A -85,B 0,C 180,E1 -7126.694,E2 -7126.694} C_VEL
LIN {X 0,Y 475.886,Z 515.692,A -85,B 0,C 180,E1 -7127.049,E2 -7127.049} C_VEL
LIN {X 0,Y 476.5,Z 499.407,A -85,B 0,C 180,E1 -7129.831,E2 -7129.831} C_VEL
LIN {X 0,Y 477.344,Z 482.813,A -85,B 0,C 180,E1 -7132.737,E2 -7132.737} C_VEL
LIN {X 0,Y 477.571,Z 477.161,A -85,B 0,C 180,E1 -7133.739,E2 -7133.739} C_VEL
LIN {X 0,Y 475.101,Z 464.889,A -85,B 0,C 180,E1 -7136.12,E2 -7136.12} C_VEL
LIN {X 0,Y 474.697,Z 462.984,A -85,B 0,C 180,E1 -7136.548,E2 -7136.548} C_VEL
LIN {X 0,Y 474.628,Z 462.995,A -85,B 0,C 180,E1 -7139.252,E2 -7139.252} C_VEL
LIN {X 0,Y 474.621,Z 462.988,A -85,B 0,C 180,E1 -7142.431,E2 -7142.431} C_VEL
LIN {X 0,Y 474.62,Z 462.992,A -85,B 0,C 180,E1 -7145.47,E2 -7145.47} C_VEL
LIN {X 0,Y 474.618,Z 462.985,A -85,B 0,C 180,E1 -7148.458,E2 -7148.458} C_VEL
LIN {X 0,Y 474.639,Z 462.984,A -85,B 0,C 180,E1 -7150.96,E2 -7150.96} C_VEL
LIN {X 0,Y 474.621,Z 462.986,A -85,B 0,C 180,E1 -7154.104,E2 -7154.104} C_VEL
LIN {X 0,Y 474.621,Z 462.986,A -85,B 0,C 180,E1 -7157.066,E2 -7157.066} C_VEL
LIN {X 0,Y 474.624,Z 462.985,A -85,B 0,C 180,E1 -7160.354,E2 -7160.354} C_VEL
LIN {X 0,Y 474.599,Z 462.993,A -85,B 0,C 180,E1 -7163.677,E2 -7163.677} C_VEL
LIN {X 0,Y 474.649,Z 462.982,A -85,B 0,C 180,E1 -7166.78,E2 -7166.78} C_VEL
LIN {X 0,Y 474.612,Z 462.994,A -85,B 0,C 180,E1 -7169.77,E2 -7169.77} C_VEL
LIN {X 0,Y 474.73,Z 462.976,A -85,B 0,C 180,E1 -7173.158,E2 -7173.158} C_VEL
LIN {X 0,Y 474.731,Z 463.157,A -85,B 0,C 180,E1 -7173.395,E2 -7173.395} C_VEL
LIN {X 0,Y 477.263,Z 475.358,A -85,B 0,C 180,E1 -7175.418,E2 -7175.418} C_VEL
LIN {X 0,Y 477.359,Z 480.459,A -85,B 0,C 180,E1 -7176.219,E2 -7176.219} C_VEL
LIN {X 0,Y 476.771,Z 498.952,A -85,B 0,C 180,E1 -7179.055,E2 -7179.055} C_VEL
LIN {X 0,Y 476.162,Z 519.237,A -85,B 0,C 180,E1 -7182.166,E2 -7182.166} C_VEL
LIN {X 0,Y 475.969,Z 526.83,A -85,B 0,C 180,E1 -7183.339,E2 -7183.339} C_VEL
LIN {X 0,Y 478.091,Z 540.36,A -85,B 0,C 180,E1 -7183.645,E2 -7183.645} C_VEL
LIN {X 0,Y 477.082,Z 636.998,A -85,B 0,C 180,E1 -7185.251,E2 -7185.251} C_VEL
LIN {X 0,Y 476.884,Z 648.97,A -85,B 0,C 180,E1 -7185.6,E2 -7185.6} C_VEL
LIN {X 0,Y 476.518,Z 661.53,A -85,B 0,C 180,E1 -7186.133,E2 -7186.133} C_VEL
LIN {X 0,Y 476.124,Z 674.528,A -85,B 0,C 180,E1 -7186.883,E2 -7186.883} C_VEL
LIN {X 0,Y 475.755,Z 685.876,A -85,B 0,C 180,E1 -7187.74,E2 -7187.74} C_VEL
LIN {X 0,Y 475.237,Z 697.162,A -85,B 0,C 180,E1 -7188.808,E2 -7188.808} C_VEL
LIN {X 0,Y 474.828,Z 707.016,A -85,B 0,C 180,E1 -7189.984,E2 -7189.984} C_VEL
LIN {X 0,Y 474.488,Z 715.685,A -85,B 0,C 180,E1 -7191.267,E2 -7191.267} C_VEL
LIN {X 0,Y 474.209,Z 722.593,A -85,B 0,C 180,E1 -7192.549,E2 -7192.549} C_VEL
LIN {X 0,Y 474.072,Z 728.895,A -85,B 0,C 180,E1 -7194.043,E2 -7194.043} C_VEL
LIN {X 0,Y 473.875,Z 733.019,A -85,B 0,C 180,E1 -7195.321,E2 -7195.321} C_VEL
LIN {X 0,Y 473.848,Z 736.068,A -85,B 0,C 180,E1 -7196.599,E2 -7196.599} C_VEL
LIN {X 0,Y 473.81,Z 737.565,A -85,B 0,C 180,E1 -7197.449,E2 -7197.449} C_VEL
LIN {X 0,Y 473.76,Z 738.61,A -85,B 0,C 180,E1 -7198.3,E2 -7198.3} C_VEL
LIN {X 0,Y 473.671,Z 739.531,A -85,B 0,C 180,E1 -7200,E2 -7200} C_VEL
LIN {X 0,Y 473.69,Z 739.351,A -85,B 0,C 180,E1 -7200.85,E2 -7200.85} C_VEL
LIN {X 0,Y 473.761,Z 738.765,A -85,B 0,C 180,E1 -7201.7,E2 -7201.7} C_VEL
LIN {X 0,Y 473.822,Z 737.789,A -85,B 0,C 180,E1 -7202.55,E2 -7202.55} C_VEL
LIN {X 0,Y 473.848,Z 736.388,A -85,B 0,C 180,E1 -7203.401,E2 -7203.401} C_VEL
LIN {X 0,Y 473.905,Z 733.456,A -85,B 0,C 180,E1 -7204.678,E2 -7204.678} C_VEL
LIN {X 0,Y 474.082,Z 729.451,A -85,B 0,C 180,E1 -7205.956,E2 -7205.956} C_VEL
LIN {X 0,Y 474.202,Z 723.272,A -85,B 0,C 180,E1 -7207.451,E2 -7207.451} C_VEL
LIN {X 0,Y 474.534,Z 716.497,A -85,B 0,C 180,E1 -7208.731,E2 -7208.731} C_VEL
LIN {X 0,Y 474.79,Z 707.979,A -85,B 0,C 180,E1 -7210.016,E2 -7210.016} C_VEL
LIN {X 0,Y 475.154,Z 699.227,A -85,B 0,C 180,E1 -7211.086,E2 -7211.086} C_VEL
LIN {X 0,Y 475.635,Z 689.61,A -85,B 0,C 180,E1 -7212.047,E2 -7212.047} C_VEL
LIN {X 0,Y 475.994,Z 678.089,A -85,B 0,C 180,E1 -7212.969,E2 -7212.969} C_VEL
LIN {X 0,Y 476.302,Z 667.243,A -85,B 0,C 180,E1 -7213.656,E2 -7213.656} C_VEL
LIN {X 0,Y 476.695,Z 655.144,A -85,B 0,C 180,E1 -7214.242,E2 -7214.242} C_VEL
LIN {X 0,Y 477.018,Z 641.8,A -85,B 0,C 180,E1 -7214.696,E2 -7214.696} C_VEL
LIN {X 0,Y 477.192,Z 627.631,A -85,B 0,C 180,E1 -7214.99,E2 -7214.99} C_VEL
LIN {X 0,Y 478.166,Z 539.818,A -85,B 0,C 180,E1 -7216.486,E2 -7216.486} C_VEL
LIN {X 0,Y 476.178,Z 528.116,A -85,B 0,C 180,E1 -7216.787,E2 -7216.787} C_VEL
LIN {X 0,Y 476.683,Z 507.844,A -85,B 0,C 180,E1 -7219.822,E2 -7219.822} C_VEL
LIN {X 0,Y 477.19,Z 488.092,A -85,B 0,C 180,E1 -7222.743,E2 -7222.743} C_VEL
LIN {X 0,Y 477.476,Z 477.048,A -85,B 0,C 180,E1 -7224.339,E2 -7224.339} C_VEL
LIN {X 0,Y 475.622,Z 466.814,A -85,B 0,C 180,E1 -7225.939,E2 -7225.939} C_VEL
LIN {X 0,Y 474.711,Z 462.981,A -85,B 0,C 180,E1 -7226.546,E2 -7226.546} C_VEL
LIN {X 0,Y 474.626,Z 462.991,A -85,B 0,C 180,E1 -7229.252,E2 -7229.252} C_VEL
LIN {X 0,Y 474.62,Z 462.993,A -85,B 0,C 180,E1 -7232.43,E2 -7232.43} C_VEL
LIN {X 0,Y 474.625,Z 462.989,A -85,B 0,C 180,E1 -7235.47,E2 -7235.47} C_VEL
LIN {X 0,Y 474.616,Z 462.989,A -85,B 0,C 180,E1 -7238.457,E2 -7238.457} C_VEL
LIN {X 0,Y 474.632,Z 462.986,A -85,B 0,C 180,E1 -7240.959,E2 -7240.959} C_VEL
LIN {X 0,Y 474.61,Z 462.993,A -85,B 0,C 180,E1 -7244.105,E2 -7244.105} C_VEL
LIN {X 0,Y 474.619,Z 462.988,A -85,B 0,C 180,E1 -7247.065,E2 -7247.065} C_VEL
LIN {X 0,Y 474.622,Z 462.986,A -85,B 0,C 180,E1 -7250.353,E2 -7250.353} C_VEL
LIN {X 0,Y 474.593,Z 462.994,A -85,B 0,C 180,E1 -7253.676,E2 -7253.676} C_VEL
LIN {X 0,Y 474.647,Z 462.986,A -85,B 0,C 180,E1 -7256.779,E2 -7256.779} C_VEL
LIN {X 0,Y 474.61,Z 462.993,A -85,B 0,C 180,E1 -7259.769,E2 -7259.769} C_VEL
LIN {X 0,Y 474.703,Z 463.039,A -85,B 0,C 180,E1 -7261.54,E2 -7261.54} C_VEL
LIN {X 0,Y 478.7,Z 479.519,A -85,B 0,C 180,E1 -7264.101,E2 -7264.101} C_VEL
LIN {X 0,Y 479.129,Z 482.921,A -85,B 0,C 180,E1 -7264.592,E2 -7264.592} C_VEL
LIN {X 0,Y 477.762,Z 507.045,A -85,B 0,C 180,E1 -7267.808,E2 -7267.808} C_VEL
LIN {X 0,Y 476.993,Z 522.928,A -85,B 0,C 180,E1 -7269.927,E2 -7269.927} C_VEL
LIN {X 0,Y 479.573,Z 540.504,A -85,B 0,C 180,E1 -7270.322,E2 -7270.322} C_VEL
LIN {X 0,Y 478.26,Z 659.674,A -85,B 0,C 180,E1 -7272.246,E2 -7272.246} C_VEL
LIN {X 0,Y 477.885,Z 674.085,A -85,B 0,C 180,E1 -7272.646,E2 -7272.646} C_VEL
LIN {X 0,Y 477.482,Z 687.109,A -85,B 0,C 180,E1 -7273.164,E2 -7273.164} C_VEL
LIN {X 0,Y 476.943,Z 700.2,A -85,B 0,C 180,E1 -7273.85,E2 -7273.85} C_VEL
LIN {X 0,Y 476.39,Z 713.081,A -85,B 0,C 180,E1 -7274.709,E2 -7274.709} C_VEL
LIN {X 0,Y 475.799,Z 724.828,A -85,B 0,C 180,E1 -7275.675,E2 -7275.675} C_VEL
LIN {X 0,Y 475.295,Z 735.615,A -85,B 0,C 180,E1 -7276.749,E2 -7276.749} C_VEL
LIN {X 0,Y 474.884,Z 746.345,A -85,B 0,C 180,E1 -7278.041,E2 -7278.041} C_VEL
LIN {X 0,Y 474.47,Z 755.172,A -85,B 0,C 180,E1 -7279.329,E2 -7279.329} C_VEL
LIN {X 0,Y 474.163,Z 763.584,A -85,B 0,C 180,E1 -7280.831,E2 -7280.831} C_VEL
LIN {X 0,Y 473.933,Z 770.336,A -85,B 0,C 180,E1 -7282.329,E2 -7282.329} C_VEL
LIN {X 0,Y 473.895,Z 774.735,A -85,B 0,C 180,E1 -7283.53,E2 -7283.53} C_VEL
LIN {X 0,Y 473.829,Z 778.683,A -85,B 0,C 180,E1 -7284.893,E2 -7284.893} C_VEL
LIN {X 0,Y 473.81,Z 782.26,A -85,B 0,C 180,E1 -7286.597,E2 -7286.597} C_VEL
LIN {X 0,Y 473.756,Z 784.377,A -85,B 0,C 180,E1 -7288.299,E2 -7288.299} C_VEL
LIN {X 0,Y 473.667,Z 785.079,A -85,B 0,C 180,E1 -7289.999,E2 -7289.999} C_VEL
LIN {X 0,Y 473.756,Z 784.381,A -85,B 0,C 180,E1 -7291.699,E2 -7291.699} C_VEL
LIN {X 0,Y 473.809,Z 782.271,A -85,B 0,C 180,E1 -7293.4,E2 -7293.4} C_VEL
LIN {X 0,Y 473.829,Z 778.698,A -85,B 0,C 180,E1 -7295.105,E2 -7295.105} C_VEL
LIN {X 0,Y 473.89,Z 773.555,A -85,B 0,C 180,E1 -7296.813,E2 -7296.813} C_VEL
LIN {X 0,Y 473.996,Z 768.569,A -85,B 0,C 180,E1 -7298.096,E2 -7298.096} C_VEL
LIN {X 0,Y 474.252,Z 761.357,A -85,B 0,C 180,E1 -7299.596,E2 -7299.596} C_VEL
LIN {X 0,Y 474.598,Z 752.398,A -85,B 0,C 180,E1 -7301.098,E2 -7301.098} C_VEL
LIN {X 0,Y 474.987,Z 742.663,A -85,B 0,C 180,E1 -7302.433,E2 -7302.433} C_VEL
LIN {X 0,Y 475.514,Z 731.594,A -85,B 0,C 180,E1 -7303.677,E2 -7303.677} C_VEL
LIN {X 0,Y 476.041,Z 719.93,A -85,B 0,C 180,E1 -7304.753,E2 -7304.753} C_VEL
LIN {X 0,Y 476.631,Z 707.033,A -85,B 0,C 180,E1 -7305.719,E2 -7305.719} C_VEL
LIN {X 0,Y 477.165,Z 694.502,A -85,B 0,C 180,E1 -7306.47,E2 -7306.47} C_VEL
LIN {X 0,Y 477.671,Z 680.662,A -85,B 0,C 180,E1 -7307.112,E2 -7307.112} C_VEL
LIN {X 0,Y 478.076,Z 666.325,A -85,B 0,C 180,E1 -7307.593,E2 -7307.593} C_VEL
LIN {X 0,Y 478.456,Z 650.96,A -85,B 0,C 180,E1 -7307.91,E2 -7307.91} C_VEL
LIN {X 0,Y 479.455,Z 539.241,A -85,B 0,C 180,E1 -7309.701,E2 -7309.701} C_VEL
LIN {X 0,Y 477.029,Z 522.798,A -85,B 0,C 180,E1 -7310.083,E2 -7310.083} C_VEL
LIN {X 0,Y 478.249,Z 498.111,A -85,B 0,C 180,E1 -7313.375,E2 -7313.375} C_VEL
LIN {X 0,Y 479.118,Z 482.918,A -85,B 0,C 180,E1 -7315.406,E2 -7315.406} C_VEL
LIN {X 0,Y 478.293,Z 477.84,A -85,B 0,C 180,E1 -7316.155,E2 -7316.155} C_VEL
LIN {X 0,Y 474.665,Z 462.984,A -85,B 0,C 180,E1 -7318.491,E2 -7318.491} C_VEL
LIN {X 0,Y 474.599,Z 462.992,A -85,B 0,C 180,E1 -7321.216,E2 -7321.216} C_VEL
LIN {X 0,Y 474.629,Z 462.981,A -85,B 0,C 180,E1 -7324.24,E2 -7324.24} C_VEL
LIN {X 0,Y 474.589,Z 462.991,A -85,B 0,C 180,E1 -7327.382,E2 -7327.382} C_VEL
LIN {X 0,Y 474.649,Z 462.983,A -85,B 0,C 180,E1 -7329.651,E2 -7329.651} C_VEL
LIN {X 0,Y 474.645,Z 462.987,A -85,B 0,C 180,E1 -7332.929,E2 -7332.929} C_VEL
LIN {X 0,Y 474.61,Z 462.986,A -85,B 0,C 180,E1 -7335.895,E2 -7335.895} C_VEL
LIN {X 0,Y 474.637,Z 462.985,A -85,B 0,C 180,E1 -7339.037,E2 -7339.037} C_VEL
LIN {X 0,Y 474.611,Z 462.984,A -85,B 0,C 180,E1 -7341.702,E2 -7341.702} C_VEL
LIN {X 0,Y 474.621,Z 462.98,A -85,B 0,C 180,E1 -7344.725,E2 -7344.725} C_VEL
LIN {X 0,Y 474.628,Z 462.983,A -85,B 0,C 180,E1 -7347.787,E2 -7347.787} C_VEL
LIN {X 0,Y 474.622,Z 462.988,A -85,B 0,C 180,E1 -7350.882,E2 -7350.882} C_VEL
LIN {X 0,Y 474.656,Z 462.981,A -85,B 0,C 180,E1 -7353.628,E2 -7353.628} C_VEL
LIN {X 0,Y 474.625,Z 462.979,A -85,B 0,C 180,E1 -7356.641,E2 -7356.641} C_VEL
LIN {X 0,Y 474.646,Z 462.978,A -85,B 0,C 180,E1 -7360.089,E2 -7360.089} C_VEL
LIN {X 0,Y 474.64,Z 462.987,A -85,B 0,C 180,E1 -7362.774,E2 -7362.774} C_VEL
LIN {X 0,Y 474.638,Z 462.983,A -85,B 0,C 180,E1 -7365.421,E2 -7365.421} C_VEL
LIN {X 0,Y 474.727,Z 462.972,A -85,B 0,C 180,E1 -7368.038,E2 -7368.038} C_VEL
LIN {X 0,Y 474.718,Z 462.973,A -85,B 0,C 180,E1 -7371.486,E2 -7371.486} C_VEL
LIN {X 0,Y 474.773,Z 462.962,A -85,B 0,C 180,E1 -7374.052,E2 -7374.052} C_VEL
LIN {X 0,Y 474.885,Z 462.95,A -85,B 0,C 180,E1 -7377.455,E2 -7377.455} C_VEL
LIN {X 0,Y 474.866,Z 462.959,A -85,B 0,C 180,E1 -7380.848,E2 -7380.848} C_VEL
LIN {X 0,Y 474.885,Z 462.956,A -85,B 0,C 180,E1 -7382.545,E2 -7382.545} C_VEL
LIN {X 0,Y 474.769,Z 462.968,A -85,B 0,C 180,E1 -7385.948,E2 -7385.948} C_VEL
LIN {X 0,Y 474.718,Z 462.975,A -85,B 0,C 180,E1 -7388.514,E2 -7388.514} C_VEL
LIN {X 0,Y 474.728,Z 462.973,A -85,B 0,C 180,E1 -7391.962,E2 -7391.962} C_VEL
LIN {X 0,Y 474.691,Z 462.977,A -85,B 0,C 180,E1 -7395.778,E2 -7395.778} C_VEL
LIN {X 0,Y 474.655,Z 462.983,A -85,B 0,C 180,E1 -7399.011,E2 -7399.011} C_VEL
LIN {X 0,Y 474.58,Z 462.989,A -85,B 0,C 180,E1 -7401.73,E2 -7401.73} C_VEL
LIN {X 0,Y 474.649,Z 462.989,A -85,B 0,C 180,E1 -7404.494,E2 -7404.494} C_VEL
LIN {X 0,Y 474.689,Z 462.976,A -85,B 0,C 180,E1 -7407.34,E2 -7407.34} C_VEL
LIN {X 0,Y 474.601,Z 462.991,A -85,B 0,C 180,E1 -7410.812,E2 -7410.812} C_VEL
LIN {X 0,Y 474.63,Z 462.984,A -85,B 0,C 180,E1 -7413.985,E2 -7413.985} C_VEL
LIN {X 0,Y 474.569,Z 462.993,A -85,B 0,C 180,E1 -7416.901,E2 -7416.901} C_VEL
LIN {X 0,Y 474.648,Z 462.982,A -85,B 0,C 180,E1 -7419.653,E2 -7419.653} C_VEL
LIN {X 0,Y 474.608,Z 462.989,A -85,B 0,C 180,E1 -7422.935,E2 -7422.935} C_VEL
LIN {X 0,Y 474.612,Z 462.988,A -85,B 0,C 180,E1 -7425.898,E2 -7425.898} C_VEL
LIN {X 0,Y 474.64,Z 462.985,A -85,B 0,C 180,E1 -7429.04,E2 -7429.04} C_VEL
LIN {X 0,Y 474.615,Z 462.988,A -85,B 0,C 180,E1 -7431.704,E2 -7431.704} C_VEL
LIN {X 0,Y 474.627,Z 462.99,A -85,B 0,C 180,E1 -7434.728,E2 -7434.728} C_VEL
LIN {X 0,Y 474.635,Z 462.987,A -85,B 0,C 180,E1 -7437.789,E2 -7437.789} C_VEL
LIN {X 0,Y 474.63,Z 462.988,A -85,B 0,C 180,E1 -7440.884,E2 -7440.884} C_VEL
LIN {X 0,Y 474.711,Z 463.031,A -85,B 0,C 180,E1 -7443.603,E2 -7443.603} C_VEL
LIN {X 0,Y 477.514,Z 476.808,A -85,B 0,C 180,E1 -7446.286,E2 -7446.286} C_VEL
LIN {X 0,Y 477.069,Z 488.694,A -85,B 0,C 180,E1 -7448.391,E2 -7448.391} C_VEL
LIN {X 0,Y 476.799,Z 493.87,A -85,B 0,C 180,E1 -7449.297,E2 -7449.297} C_VEL
LIN {X 0,Y 475.969,Z 497.32,A -85,B 0,C 180,E1 -7449.866,E2 -7449.866} C_VEL
LIN {X 0,Y 469.876,Z 509.162,A -85,B 0,C 180,E1 -7451.653,E2 -7451.653} C_VEL
LIN {X 0,Y 469.087,Z 512.669,A -85,B 0,C 180,E1 -7452.228,E2 -7452.228} C_VEL
LIN {X 0,Y 468.972,Z 515.701,A -85,B 0,C 180,E1 -7452.75,E2 -7452.75} C_VEL
LIN {X 0,Y 472.004,Z 532.335,A -85,B 0,C 180,E1 -7453.14,E2 -7453.14} C_VEL
LIN {X 0,Y 471.467,Z 626.619,A -85,B 0,C 180,E1 -7454.492,E2 -7454.492} C_VEL
LIN {X 0,Y 471.221,Z 639.429,A -85,B 0,C 180,E1 -7454.844,E2 -7454.844} C_VEL
LIN {X 0,Y 470.804,Z 651.846,A -85,B 0,C 180,E1 -7455.356,E2 -7455.356} C_VEL
LIN {X 0,Y 470.318,Z 664.231,A -85,B 0,C 180,E1 -7456.058,E2 -7456.058} C_VEL
LIN {X 0,Y 469.799,Z 675.828,A -85,B 0,C 180,E1 -7456.929,E2 -7456.929} C_VEL
LIN {X 0,Y 469.113,Z 686.12,A -85,B 0,C 180,E1 -7457.894,E2 -7457.894} C_VEL
LIN {X 0,Y 468.628,Z 695.425,A -85,B 0,C 180,E1 -7458.978,E2 -7458.978} C_VEL
LIN {X 0,Y 468.177,Z 703.05,A -85,B 0,C 180,E1 -7460.06,E2 -7460.06} C_VEL
LIN {X 0,Y 467.687,Z 710.526,A -85,B 0,C 180,E1 -7461.359,E2 -7461.359} C_VEL
LIN {X 0,Y 467.315,Z 716.529,A -85,B 0,C 180,E1 -7462.657,E2 -7462.657} C_VEL
LIN {X 0,Y 467.068,Z 721.312,A -85,B 0,C 180,E1 -7463.955,E2 -7463.955} C_VEL
LIN {X 0,Y 466.924,Z 725.027,A -85,B 0,C 180,E1 -7465.253,E2 -7465.253} C_VEL
LIN {X 0,Y 466.844,Z 727.777,A -85,B 0,C 180,E1 -7466.549,E2 -7466.549} C_VEL
LIN {X 0,Y 466.823,Z 729.081,A -85,B 0,C 180,E1 -7467.413,E2 -7467.413} C_VEL
LIN {X 0,Y 466.622,Z 730.601,A -85,B 0,C 180,E1 -7469.138,E2 -7469.138} C_VEL
LIN {X 0,Y 466.622,Z 730.647,A -85,B 0,C 180,E1 -7470.864,E2 -7470.864} C_VEL
LIN {X 0,Y 466.82,Z 729.187,A -85,B 0,C 180,E1 -7472.59,E2 -7472.59} C_VEL
LIN {X 0,Y 466.939,Z 726.244,A -85,B 0,C 180,E1 -7474.317,E2 -7474.317} C_VEL
LIN {X 0,Y 466.936,Z 722.947,A -85,B 0,C 180,E1 -7475.616,E2 -7475.616} C_VEL
LIN {X 0,Y 467.204,Z 718.604,A -85,B 0,C 180,E1 -7476.913,E2 -7476.913} C_VEL
LIN {X 0,Y 467.596,Z 712.039,A -85,B 0,C 180,E1 -7478.428,E2 -7478.428} C_VEL
LIN {X 0,Y 468.022,Z 704.927,A -85,B 0,C 180,E1 -7479.727,E2 -7479.727} C_VEL
LIN {X 0,Y 468.558,Z 696.106,A -85,B 0,C 180,E1 -7481.026,E2 -7481.026} C_VEL
LIN {X 0,Y 469.101,Z 686.963,A -85,B 0,C 180,E1 -7482.108,E2 -7482.108} C_VEL
LIN {X 0,Y 469.776,Z 675.919,A -85,B 0,C 180,E1 -7483.155,E2 -7483.155} C_VEL
LIN {X 0,Y 470.274,Z 665.491,A -85,B 0,C 180,E1 -7483.945,E2 -7483.945} C_VEL
LIN {X 0,Y 470.819,Z 653.643,A -85,B 0,C 180,E1 -7484.646,E2 -7484.646} C_VEL
LIN {X 0,Y 471.157,Z 641.148,A -85,B 0,C 180,E1 -7485.188,E2 -7485.188} C_VEL
LIN {X 0,Y 471.499,Z 628.036,A -85,B 0,C 180,E1 -7485.564,E2 -7485.564} C_VEL
LIN {X 0,Y 471.676,Z 601.248,A -85,B 0,C 180,E1 -7485.974,E2 -7485.974} C_VEL
LIN {X 0,Y 471.878,Z 531.043,A -85,B 0,C 180,E1 -7486.974,E2 -7486.974} C_VEL
LIN {X 0,Y 468.964,Z 515.718,A -85,B 0,C 180,E1 -7487.339,E2 -7487.339} C_VEL
LIN {X 0,Y 469.63,Z 499.571,A -85,B 0,C 180,E1 -7490.134,E2 -7490.134} C_VEL
LIN {X 0,Y 470.462,Z 484.234,A -85,B 0,C 180,E1 -7492.856,E2 -7492.856} C_VEL
LIN {X 0,Y 470.707,Z 479.107,A -85,B 0,C 180,E1 -7493.775,E2 -7493.775} C_VEL
LIN {X 0,Y 468.641,Z 468.414,A -85,B 0,C 180,E1 -7495.868,E2 -7495.868} C_VEL
LIN {X 0,Y 467.675,Z 463.86,A -85,B 0,C 180,E1 -7496.798,E2 -7496.798} C_VEL
LIN {X 0,Y 467.56,Z 463.876,A -85,B 0,C 180,E1 -7499.739,E2 -7499.739} C_VEL
LIN {X 0,Y 467.589,Z 463.864,A -85,B 0,C 180,E1 -7502.759,E2 -7502.759} C_VEL
LIN {X 0,Y 467.559,Z 463.869,A -85,B 0,C 180,E1 -7505.89,E2 -7505.89} C_VEL
LIN {X 0,Y 467.589,Z 463.862,A -85,B 0,C 180,E1 -7509.145,E2 -7509.145} C_VEL
LIN {X 0,Y 467.593,Z 463.862,A -85,B 0,C 180,E1 -7512.567,E2 -7512.567} C_VEL
LIN {X 0,Y 467.577,Z 463.862,A -85,B 0,C 180,E1 -7515.053,E2 -7515.053} C_VEL
LIN {X 0,Y 467.595,Z 463.864,A -85,B 0,C 180,E1 -7517.44,E2 -7517.44} C_VEL
LIN {X 0,Y 467.566,Z 463.864,A -85,B 0,C 180,E1 -7520.853,E2 -7520.853} C_VEL
LIN {X 0,Y 467.569,Z 463.865,A -85,B 0,C 180,E1 -7524.261,E2 -7524.261} C_VEL
LIN {X 0,Y 467.588,Z 463.865,A -85,B 0,C 180,E1 -7527.321,E2 -7527.321} C_VEL
LIN {X 0,Y 467.576,Z 463.865,A -85,B 0,C 180,E1 -7530.668,E2 -7530.668} C_VEL
LIN {X 0,Y 467.693,Z 463.899,A -85,B 0,C 180,E1 -7533.148,E2 -7533.148} C_VEL
LIN {X 0,Y 470.565,Z 478.185,A -85,B 0,C 180,E1 -7535.535,E2 -7535.535} C_VEL
LIN {X 0,Y 469.946,Z 497.393,A -85,B 0,C 180,E1 -7538.506,E2 -7538.506} C_VEL
LIN {X 0,Y 469.307,Z 517.845,A -85,B 0,C 180,E1 -7541.67,E2 -7541.67} C_VEL
LIN {X 0,Y 469.043,Z 527.275,A -85,B 0,C 180,E1 -7543.102,E2 -7543.102} C_VEL
LIN {X 0,Y 471.254,Z 540.652,A -85,B 0,C 180,E1 -7543.417,E2 -7543.417} C_VEL
LIN {X 0,Y 470.169,Z 637.156,A -85,B 0,C 180,E1 -7545.057,E2 -7545.057} C_VEL
LIN {X 0,Y 469.928,Z 649.907,A -85,B 0,C 180,E1 -7545.437,E2 -7545.437} C_VEL
LIN {X 0,Y 469.58,Z 662.262,A -85,B 0,C 180,E1 -7545.979,E2 -7545.979} C_VEL
LIN {X 0,Y 469.187,Z 674.329,A -85,B 0,C 180,E1 -7546.685,E2 -7546.685} C_VEL
LIN {X 0,Y 468.86,Z 684.749,A -85,B 0,C 180,E1 -7547.464,E2 -7547.464} C_VEL
LIN {X 0,Y 468.348,Z 695.081,A -85,B 0,C 180,E1 -7548.422,E2 -7548.422} C_VEL
LIN {X 0,Y 467.936,Z 705.479,A -85,B 0,C 180,E1 -7549.617,E2 -7549.617} C_VEL
LIN {X 0,Y 467.539,Z 714.481,A -85,B 0,C 180,E1 -7550.919,E2 -7550.919} C_VEL
LIN {X 0,Y 467.21,Z 721.723,A -85,B 0,C 180,E1 -7552.219,E2 -7552.219} C_VEL
LIN {X 0,Y 467.005,Z 727.905,A -85,B 0,C 180,E1 -7553.622,E2 -7553.622} C_VEL
LIN {X 0,Y 466.799,Z 732.043,A -85,B 0,C 180,E1 -7554.817,E2 -7554.817} C_VEL
LIN {X 0,Y 466.843,Z 734.412,A -85,B 0,C 180,E1 -7555.683,E2 -7555.683} C_VEL
LIN {X 0,Y 466.784,Z 736.356,A -85,B 0,C 180,E1 -7556.547,E2 -7556.547} C_VEL
LIN {X 0,Y 466.726,Z 737.872,A -85,B 0,C 180,E1 -7557.411,E2 -7557.411} C_VEL
LIN {X 0,Y 466.696,Z 738.926,A -85,B 0,C 180,E1 -7558.274,E2 -7558.274} C_VEL
LIN {X 0,Y 466.6,Z 739.863,A -85,B 0,C 180,E1 -7560,E2 -7560} C_VEL
LIN {X 0,Y 466.621,Z 739.689,A -85,B 0,C 180,E1 -7560.863,E2 -7560.863} C_VEL
LIN {X 0,Y 466.697,Z 739.104,A -85,B 0,C 180,E1 -7561.726,E2 -7561.726} C_VEL
LIN {X 0,Y 466.737,Z 738.129,A -85,B 0,C 180,E1 -7562.589,E2 -7562.589} C_VEL
LIN {X 0,Y 466.784,Z 736.725,A -85,B 0,C 180,E1 -7563.453,E2 -7563.453} C_VEL
LIN {X 0,Y 466.815,Z 733.785,A -85,B 0,C 180,E1 -7564.75,E2 -7564.75} C_VEL
LIN {X 0,Y 467.035,Z 729.764,A -85,B 0,C 180,E1 -7566.046,E2 -7566.046} C_VEL
LIN {X 0,Y 467.156,Z 723.56,A -85,B 0,C 180,E1 -7567.564,E2 -7567.564} C_VEL
LIN {X 0,Y 467.502,Z 716.756,A -85,B 0,C 180,E1 -7568.864,E2 -7568.864} C_VEL
LIN {X 0,Y 467.809,Z 708.192,A -85,B 0,C 180,E1 -7570.167,E2 -7570.167} C_VEL
LIN {X 0,Y 468.191,Z 699.41,A -85,B 0,C 180,E1 -7571.253,E2 -7571.253} C_VEL
LIN {X 0,Y 468.684,Z 689.856,A -85,B 0,C 180,E1 -7572.221,E2 -7572.221} C_VEL
LIN {X 0,Y 469.049,Z 678.982,A -85,B 0,C 180,E1 -7573.11,E2 -7573.11} C_VEL
LIN {X 0,Y 469.421,Z 667.386,A -85,B 0,C 180,E1 -7573.86,E2 -7573.86} C_VEL
LIN {X 0,Y 469.826,Z 655.245,A -85,B 0,C 180,E1 -7574.455,E2 -7574.455} C_VEL
LIN {X 0,Y 470.162,Z 641.84,A -85,B 0,C 180,E1 -7574.915,E2 -7574.915} C_VEL
LIN {X 0,Y 470.335,Z 627.51,A -85,B 0,C 180,E1 -7575.214,E2 -7575.214} C_VEL
LIN {X 0,Y 471.409,Z 540.651,A -85,B 0,C 180,E1 -7576.735,E2 -7576.735} C_VEL
LIN {X 0,Y 469.328,Z 528.48,A -85,B 0,C 180,E1 -7577.073,E2 -7577.073} C_VEL
LIN {X 0,Y 469.865,Z 508.196,A -85,B 0,C 180,E1 -7580.122,E2 -7580.122} C_VEL
LIN {X 0,Y 470.352,Z 491.413,A -85,B 0,C 180,E1 -7582.628,E2 -7582.628} C_VEL
LIN {X 0,Y 470.68,Z 478.988,A -85,B 0,C 180,E1 -7584.451,E2 -7584.451} C_VEL
LIN {X 0,Y 469.005,Z 469.381,A -85,B 0,C 180,E1 -7585.959,E2 -7585.959} C_VEL
LIN {X 0,Y 467.686,Z 463.856,A -85,B 0,C 180,E1 -7586.88,E2 -7586.88} C_VEL
LIN {X 0,Y 467.559,Z 463.873,A -85,B 0,C 180,E1 -7589.738,E2 -7589.738} C_VEL
LIN {X 0,Y 467.588,Z 463.866,A -85,B 0,C 180,E1 -7592.758,E2 -7592.758} C_VEL
LIN {X 0,Y 467.562,Z 463.87,A -85,B 0,C 180,E1 -7595.889,E2 -7595.889} C_VEL
LIN {X 0,Y 467.587,Z 463.863,A -85,B 0,C 180,E1 -7599.144,E2 -7599.144} C_VEL
LIN {X 0,Y 467.591,Z 463.864,A -85,B 0,C 180,E1 -7602.566,E2 -7602.566} C_VEL
LIN {X 0,Y 467.57,Z 463.866,A -85,B 0,C 180,E1 -7605.052,E2 -7605.052} C_VEL
LIN {X 0,Y 467.593,Z 463.864,A -85,B 0,C 180,E1 -7607.439,E2 -7607.439} C_VEL
LIN {X 0,Y 467.564,Z 463.864,A -85,B 0,C 180,E1 -7610.853,E2 -7610.853} C_VEL
LIN {X 0,Y 467.564,Z 463.867,A -85,B 0,C 180,E1 -7614.26,E2 -7614.26} C_VEL
LIN {X 0,Y 467.586,Z 463.867,A -85,B 0,C 180,E1 -7617.32,E2 -7617.32} C_VEL
LIN {X 0,Y 467.575,Z 463.87,A -85,B 0,C 180,E1 -7620.667,E2 -7620.667} C_VEL
LIN {X 0,Y 467.642,Z 463.963,A -85,B 0,C 180,E1 -7621.23,E2 -7621.23} C_VEL
LIN {X 0,Y 471.489,Z 479.627,A -85,B 0,C 180,E1 -7623.713,E2 -7623.713} C_VEL
LIN {X 0,Y 472.313,Z 484.441,A -85,B 0,C 180,E1 -7624.435,E2 -7624.435} C_VEL
LIN {X 0,Y 470.929,Z 507.288,A -85,B 0,C 180,E1 -7627.531,E2 -7627.531} C_VEL
LIN {X 0,Y 470.156,Z 523.195,A -85,B 0,C 180,E1 -7629.66,E2 -7629.66} C_VEL
LIN {X 0,Y 472.859,Z 541.863,A -85,B 0,C 180,E1 -7630.079,E2 -7630.079} C_VEL
LIN {X 0,Y 471.449,Z 659.417,A -85,B 0,C 180,E1 -7632.009,E2 -7632.009} C_VEL
LIN {X 0,Y 471.041,Z 673.778,A -85,B 0,C 180,E1 -7632.413,E2 -7632.413} C_VEL
LIN {X 0,Y 470.578,Z 687.352,A -85,B 0,C 180,E1 -7632.966,E2 -7632.966} C_VEL
LIN {X 0,Y 470.001,Z 701.185,A -85,B 0,C 180,E1 -7633.717,E2 -7633.717} C_VEL
LIN {X 0,Y 469.379,Z 713.793,A -85,B 0,C 180,E1 -7634.586,E2 -7634.586} C_VEL
LIN {X 0,Y 468.801,Z 725.341,A -85,B 0,C 180,E1 -7635.567,E2 -7635.567} C_VEL
LIN {X 0,Y 468.188,Z 736.945,A -85,B 0,C 180,E1 -7636.766,E2 -7636.766} C_VEL
LIN {X 0,Y 467.798,Z 747.302,A -85,B 0,C 180,E1 -7638.077,E2 -7638.077} C_VEL
LIN {X 0,Y 467.385,Z 755.886,A -85,B 0,C 180,E1 -7639.384,E2 -7639.384} C_VEL
LIN {X 0,Y 467.061,Z 764.085,A -85,B 0,C 180,E1 -7640.908,E2 -7640.908} C_VEL
LIN {X 0,Y 466.855,Z 769.831,A -85,B 0,C 180,E1 -7642.212,E2 -7642.212} C_VEL
LIN {X 0,Y 466.798,Z 774.667,A -85,B 0,C 180,E1 -7643.555,E2 -7643.555} C_VEL
LIN {X 0,Y 466.761,Z 778.23,A -85,B 0,C 180,E1 -7644.816,E2 -7644.816} C_VEL
LIN {X 0,Y 466.738,Z 781.83,A -85,B 0,C 180,E1 -7646.546,E2 -7646.546} C_VEL
LIN {X 0,Y 466.692,Z 783.963,A -85,B 0,C 180,E1 -7648.273,E2 -7648.273} C_VEL
LIN {X 0,Y 466.596,Z 784.671,A -85,B 0,C 180,E1 -7649.999,E2 -7649.999} C_VEL
LIN {X 0,Y 466.692,Z 783.967,A -85,B 0,C 180,E1 -7651.725,E2 -7651.725} C_VEL
LIN {X 0,Y 466.737,Z 781.839,A -85,B 0,C 180,E1 -7653.452,E2 -7653.452} C_VEL
LIN {X 0,Y 466.761,Z 778.239,A -85,B 0,C 180,E1 -7655.182,E2 -7655.182} C_VEL
LIN {X 0,Y 466.821,Z 773.064,A -85,B 0,C 180,E1 -7656.916,E2 -7656.916} C_VEL
LIN {X 0,Y 466.93,Z 768.043,A -85,B 0,C 180,E1 -7658.22,E2 -7658.22} C_VEL
LIN {X 0,Y 467.183,Z 760.794,A -85,B 0,C 180,E1 -7659.742,E2 -7659.742} C_VEL
LIN {X 0,Y 467.534,Z 751.802,A -85,B 0,C 180,E1 -7661.268,E2 -7661.268} C_VEL
LIN {X 0,Y 467.98,Z 741.854,A -85,B 0,C 180,E1 -7662.646,E2 -7662.646} C_VEL
LIN {X 0,Y 468.545,Z 730.924,A -85,B 0,C 180,E1 -7663.885,E2 -7663.885} C_VEL
LIN {X 0,Y 469.089,Z 719.217,A -85,B 0,C 180,E1 -7664.976,E2 -7664.976} C_VEL
LIN {X 0,Y 469.716,Z 706.264,A -85,B 0,C 180,E1 -7665.957,E2 -7665.957} C_VEL
LIN {X 0,Y 470.334,Z 693.073,A -85,B 0,C 180,E1 -7666.748,E2 -7666.748} C_VEL
LIN {X 0,Y 470.84,Z 679.685,A -85,B 0,C 180,E1 -7667.368,E2 -7667.368} C_VEL
LIN {X 0,Y 471.28,Z 665.014,A -85,B 0,C 180,E1 -7667.855,E2 -7667.855} C_VEL
LIN {X 0,Y 471.643,Z 649.043,A -85,B 0,C 180,E1 -7668.178,E2 -7668.178} C_VEL
LIN {X 0,Y 472.788,Z 540.651,A -85,B 0,C 180,E1 -7669.941,E2 -7669.941} C_VEL
LIN {X 0,Y 470.108,Z 522.736,A -85,B 0,C 180,E1 -7670.366,E2 -7670.366} C_VEL
LIN {X 0,Y 471.391,Z 499.603,A -85,B 0,C 180,E1 -7673.503,E2 -7673.503} C_VEL
LIN {X 0,Y 472.293,Z 484.433,A -85,B 0,C 180,E1 -7675.564,E2 -7675.564} C_VEL
LIN {X 0,Y 471.481,Z 479.633,A -85,B 0,C 180,E1 -7676.285,E2 -7676.285} C_VEL
LIN {X 0,Y 467.61,Z 463.862,A -85,B 0,C 180,E1 -7678.794,E2 -7678.794} C_VEL
LIN {X 0,Y 467.581,Z 463.864,A -85,B 0,C 180,E1 -7681.739,E2 -7681.739} C_VEL
LIN {X 0,Y 467.563,Z 463.856,A -85,B 0,C 180,E1 -7684.831,E2 -7684.831} C_VEL
LIN {X 0,Y 467.567,Z 463.866,A -85,B 0,C 180,E1 -7688.042,E2 -7688.042} C_VEL
LIN {X 0,Y 467.591,Z 463.865,A -85,B 0,C 180,E1 -7690.261,E2 -7690.261} C_VEL
LIN {X 0,Y 467.612,Z 463.864,A -85,B 0,C 180,E1 -7692.57,E2 -7692.57} C_VEL
LIN {X 0,Y 467.567,Z 463.865,A -85,B 0,C 180,E1 -7696.175,E2 -7696.175} C_VEL
LIN {X 0,Y 467.581,Z 463.868,A -85,B 0,C 180,E1 -7698.721,E2 -7698.721} C_VEL
LIN {X 0,Y 467.569,Z 463.862,A -85,B 0,C 180,E1 -7701.406,E2 -7701.406} C_VEL
LIN {X 0,Y 467.554,Z 463.857,A -85,B 0,C 180,E1 -7704.259,E2 -7704.259} C_VEL
LIN {X 0,Y 467.572,Z 463.862,A -85,B 0,C 180,E1 -7707.32,E2 -7707.32} C_VEL
LIN {X 0,Y 467.569,Z 463.87,A -85,B 0,C 180,E1 -7710.665,E2 -7710.665} C_VEL
LIN {X 0,Y 467.617,Z 463.859,A -85,B 0,C 180,E1 -7713.2,E2 -7713.2} C_VEL
LIN {X 0,Y 467.582,Z 463.859,A -85,B 0,C 180,E1 -7716.467,E2 -7716.467} C_VEL
LIN {X 0,Y 467.613,Z 463.852,A -85,B 0,C 180,E1 -7719.777,E2 -7719.777} C_VEL
LIN {X 0,Y 467.598,Z 463.867,A -85,B 0,C 180,E1 -7722.506,E2 -7722.506} C_VEL
LIN {X 0,Y 467.596,Z 463.861,A -85,B 0,C 180,E1 -7725.196,E2 -7725.196} C_VEL
LIN {X 0,Y 467.686,Z 463.848,A -85,B 0,C 180,E1 -7727.855,E2 -7727.855} C_VEL
LIN {X 0,Y 467.672,Z 463.851,A -85,B 0,C 180,E1 -7731.357,E2 -7731.357} C_VEL
LIN {X 0,Y 467.737,Z 463.838,A -85,B 0,C 180,E1 -7733.963,E2 -7733.963} C_VEL
LIN {X 0,Y 467.85,Z 463.826,A -85,B 0,C 180,E1 -7737.417,E2 -7737.417} C_VEL
LIN {X 0,Y 467.871,Z 463.825,A -85,B 0,C 180,E1 -7740,E2 -7740} C_VEL
LIN {X 0,Y 467.85,Z 463.831,A -85,B 0,C 180,E1 -7742.583,E2 -7742.583} C_VEL
LIN {X 0,Y 467.733,Z 463.845,A -85,B 0,C 180,E1 -7746.038,E2 -7746.038} C_VEL
LIN {X 0,Y 467.672,Z 463.853,A -85,B 0,C 180,E1 -7748.643,E2 -7748.643} C_VEL
LIN {X 0,Y 467.672,Z 463.854,A -85,B 0,C 180,E1 -7752.145,E2 -7752.145} C_VEL
LIN {X 0,Y 467.656,Z 463.854,A -85,B 0,C 180,E1 -7755.893,E2 -7755.893} C_VEL
LIN {X 0,Y 467.613,Z 463.858,A -85,B 0,C 180,E1 -7759.308,E2 -7759.308} C_VEL
LIN {X 0,Y 467.525,Z 463.87,A -85,B 0,C 180,E1 -7762.074,E2 -7762.074} C_VEL
LIN {X 0,Y 467.593,Z 463.863,A -85,B 0,C 180,E1 -7764.888,E2 -7764.888} C_VEL
LIN {X 0,Y 467.619,Z 463.857,A -85,B 0,C 180,E1 -7767.769,E2 -7767.769} C_VEL
LIN {X 0,Y 467.564,Z 463.866,A -85,B 0,C 180,E1 -7771.047,E2 -7771.047} C_VEL
LIN {X 0,Y 467.582,Z 463.864,A -85,B 0,C 180,E1 -7774.244,E2 -7774.244} C_VEL
LIN {X 0,Y 467.544,Z 463.866,A -85,B 0,C 180,E1 -7777.188,E2 -7777.188} C_VEL
LIN {X 0,Y 467.589,Z 463.866,A -85,B 0,C 180,E1 -7780.264,E2 -7780.264} C_VEL
LIN {X 0,Y 467.579,Z 463.868,A -85,B 0,C 180,E1 -7782.568,E2 -7782.568} C_VEL
LIN {X 0,Y 467.564,Z 463.866,A -85,B 0,C 180,E1 -7785.054,E2 -7785.054} C_VEL
LIN {X 0,Y 467.618,Z 463.858,A -85,B 0,C 180,E1 -7787.445,E2 -7787.445} C_VEL
LIN {X 0,Y 467.614,Z 463.862,A -85,B 0,C 180,E1 -7790.86,E2 -7790.86} C_VEL
LIN {X 0,Y 467.559,Z 463.868,A -85,B 0,C 180,E1 -7794.262,E2 -7794.262} C_VEL
LIN {X 0,Y 467.579,Z 463.865,A -85,B 0,C 180,E1 -7797.322,E2 -7797.322} C_VEL
LIN {X 0,Y 467.576,Z 463.866,A -85,B 0,C 180,E1 -7800.667,E2 -7800.667} C_VEL
LIN {X 0,Y 467.681,Z 463.956,A -85,B 0,C 180,E1 -7803.326,E2 -7803.326} C_VEL
LIN {X 0,Y 470.414,Z 476.956,A -85,B 0,C 180,E1 -7805.907,E2 -7805.907} C_VEL
LIN {X 0,Y 470.656,Z 481.171,A -85,B 0,C 180,E1 -7806.691,E2 -7806.691} C_VEL
LIN {X 0,Y 469.744,Z 497.787,A -85,B 0,C 180,E1 -7809.645,E2 -7809.645} C_VEL
LIN {X 0,Y 469.087,Z 512.669,A -85,B 0,C 180,E1 -7812.228,E2 -7812.228} C_VEL
LIN {X 0,Y 468.537,Z 514.682,A -85,B 0,C 180,E1 -7812.455,E2 -7812.455} C_VEL
LIN {X 0,Y 466.943,Z 517.933,A -85,B 0,C 180,E1 -7812.616,E2 -7812.616} C_VEL
LIN {X 0,Y 464.595,Z 522.499,A -85,B 0,C 180,E1 -7812.672,E2 -7812.672} C_VEL
LIN {X 0,Y 463.266,Z 526.985,A -85,B 0,C 180,E1 -7812.697,E2 -7812.697} C_VEL
LIN {X 0,Y 463.258,Z 530.735,A -85,B 0,C 180,E1 -7812.753,E2 -7812.753} C_VEL
LIN {X 0,Y 465.193,Z 542.439,A -85,B 0,C 180,E1 -7813.009,E2 -7813.009} C_VEL
LIN {X 0,Y 465.216,Z 543.526,A -85,B 0,C 180,E1 -7813.026,E2 -7813.026} C_VEL
LIN {X 0,Y 464.71,Z 626.775,A -85,B 0,C 180,E1 -7814.233,E2 -7814.233} C_VEL
LIN {X 0,Y 464.451,Z 639.65,A -85,B 0,C 180,E1 -7814.59,E2 -7814.59} C_VEL
LIN {X 0,Y 463.993,Z 652.668,A -85,B 0,C 180,E1 -7815.136,E2 -7815.136} C_VEL
LIN {X 0,Y 463.468,Z 664.915,A -85,B 0,C 180,E1 -7815.848,E2 -7815.848} C_VEL
LIN {X 0,Y 462.929,Z 676.485,A -85,B 0,C 180,E1 -7816.735,E2 -7816.735} C_VEL
LIN {X 0,Y 462.204,Z 686.693,A -85,B 0,C 180,E1 -7817.71,E2 -7817.71} C_VEL
LIN {X 0,Y 461.694,Z 695.962,A -85,B 0,C 180,E1 -7818.81,E2 -7818.81} C_VEL
LIN {X 0,Y 461.201,Z 703.561,A -85,B 0,C 180,E1 -7819.908,E2 -7819.908} C_VEL
LIN {X 0,Y 460.679,Z 711.005,A -85,B 0,C 180,E1 -7821.226,E2 -7821.226} C_VEL
LIN {X 0,Y 460.292,Z 716.989,A -85,B 0,C 180,E1 -7822.544,E2 -7822.544} C_VEL
LIN {X 0,Y 460.031,Z 721.756,A -85,B 0,C 180,E1 -7823.862,E2 -7823.862} C_VEL
LIN {X 0,Y 459.867,Z 725.458,A -85,B 0,C 180,E1 -7825.18,E2 -7825.18} C_VEL
LIN {X 0,Y 459.78,Z 728.198,A -85,B 0,C 180,E1 -7826.496,E2 -7826.496} C_VEL
LIN {X 0,Y 459.751,Z 729.497,A -85,B 0,C 180,E1 -7827.373,E2 -7827.373} C_VEL
LIN {X 0,Y 459.555,Z 731.01,A -85,B 0,C 180,E1 -7829.125,E2 -7829.125} C_VEL
LIN {X 0,Y 459.555,Z 731.056,A -85,B 0,C 180,E1 -7830.877,E2 -7830.877} C_VEL
LIN {X 0,Y 459.747,Z 729.602,A -85,B 0,C 180,E1 -7832.63,E2 -7832.63} C_VEL
LIN {X 0,Y 459.886,Z 726.67,A -85,B 0,C 180,E1 -7834.383,E2 -7834.383} C_VEL
LIN {X 0,Y 459.893,Z 723.382,A -85,B 0,C 180,E1 -7835.702,E2 -7835.702} C_VEL
LIN {X 0,Y 460.178,Z 719.052,A -85,B 0,C 180,E1 -7837.019,E2 -7837.019} C_VEL
LIN {X 0,Y 460.583,Z 712.512,A -85,B 0,C 180,E1 -7838.557,E2 -7838.557} C_VEL
LIN {X 0,Y 461.046,Z 705.421,A -85,B 0,C 180,E1 -7839.876,E2 -7839.876} C_VEL
LIN {X 0,Y 461.611,Z 696.626,A -85,B 0,C 180,E1 -7841.194,E2 -7841.194} C_VEL
LIN {X 0,Y 462.288,Z 686.477,A -85,B 0,C 180,E1 -7842.401,E2 -7842.401} C_VEL
LIN {X 0,Y 462.981,Z 675.616,A -85,B 0,C 180,E1 -7843.431,E2 -7843.431} C_VEL
LIN {X 0,Y 463.461,Z 664.59,A -85,B 0,C 180,E1 -7844.267,E2 -7844.267} C_VEL
LIN {X 0,Y 464.066,Z 652.204,A -85,B 0,C 180,E1 -7844.976,E2 -7844.976} C_VEL
LIN {X 0,Y 464.448,Z 639.793,A -85,B 0,C 180,E1 -7845.497,E2 -7845.497} C_VEL
LIN {X 0,Y 464.771,Z 626.967,A -85,B 0,C 180,E1 -7845.852,E2 -7845.852} C_VEL
LIN {X 0,Y 465.165,Z 531.967,A -85,B 0,C 180,E1 -7847.238,E2 -7847.238} C_VEL
LIN {X 0,Y 462.066,Z 515.735,A -85,B 0,C 180,E1 -7847.638,E2 -7847.638} C_VEL
LIN {X 0,Y 462.72,Z 501.016,A -85,B 0,C 180,E1 -7850.215,E2 -7850.215} C_VEL
LIN {X 0,Y 463.593,Z 485.778,A -85,B 0,C 180,E1 -7852.955,E2 -7852.955} C_VEL
LIN {X 0,Y 463.81,Z 480.522,A -85,B 0,C 180,E1 -7853.913,E2 -7853.913} C_VEL
LIN {X 0,Y 461.544,Z 469.022,A -85,B 0,C 180,E1 -7856.206,E2 -7856.206} C_VEL
LIN {X 0,Y 460.606,Z 464.742,A -85,B 0,C 180,E1 -7857.12,E2 -7857.12} C_VEL
LIN {X 0,Y 460.517,Z 464.752,A -85,B 0,C 180,E1 -7860.241,E2 -7860.241} C_VEL
LIN {X 0,Y 460.535,Z 464.746,A -85,B 0,C 180,E1 -7863.325,E2 -7863.325} C_VEL
LIN {X 0,Y 460.482,Z 464.747,A -85,B 0,C 180,E1 -7866.53,E2 -7866.53} C_VEL
LIN {X 0,Y 460.565,Z 464.742,A -85,B 0,C 180,E1 -7869.86,E2 -7869.86} C_VEL
LIN {X 0,Y 460.523,Z 464.743,A -85,B 0,C 180,E1 -7872.901,E2 -7872.901} C_VEL
LIN {X 0,Y 460.517,Z 464.749,A -85,B 0,C 180,E1 -7875.831,E2 -7875.831} C_VEL
LIN {X 0,Y 460.536,Z 464.739,A -85,B 0,C 180,E1 -7878.989,E2 -7878.989} C_VEL
LIN {X 0,Y 460.534,Z 464.737,A -85,B 0,C 180,E1 -7882.38,E2 -7882.38} C_VEL
LIN {X 0,Y 460.555,Z 464.745,A -85,B 0,C 180,E1 -7885.624,E2 -7885.624} C_VEL
LIN {X 0,Y 460.543,Z 464.74,A -85,B 0,C 180,E1 -7888.745,E2 -7888.745} C_VEL
LIN {X 0,Y 460.587,Z 464.738,A -85,B 0,C 180,E1 -7892.254,E2 -7892.254} C_VEL
LIN {X 0,Y 460.683,Z 464.918,A -85,B 0,C 180,E1 -7892.947,E2 -7892.947} C_VEL
LIN {X 0,Y 463.667,Z 479.655,A -85,B 0,C 180,E1 -7895.43,E2 -7895.43} C_VEL
LIN {X 0,Y 463.04,Z 498.855,A -85,B 0,C 180,E1 -7898.421,E2 -7898.421} C_VEL
LIN {X 0,Y 462.371,Z 519.393,A -85,B 0,C 180,E1 -7901.615,E2 -7901.615} C_VEL
LIN {X 0,Y 462.151,Z 527.585,A -85,B 0,C 180,E1 -7902.859,E2 -7902.859} C_VEL
LIN {X 0,Y 464.427,Z 541.525,A -85,B 0,C 180,E1 -7903.194,E2 -7903.194} C_VEL
LIN {X 0,Y 463.266,Z 637.307,A -85,B 0,C 180,E1 -7904.857,E2 -7904.857} C_VEL
LIN {X 0,Y 463.083,Z 649.32,A -85,B 0,C 180,E1 -7905.217,E2 -7905.217} C_VEL
LIN {X 0,Y 462.669,Z 661.939,A -85,B 0,C 180,E1 -7905.765,E2 -7905.765} C_VEL
LIN {X 0,Y 462.239,Z 674.779,A -85,B 0,C 180,E1 -7906.525,E2 -7906.525} C_VEL
LIN {X 0,Y 461.857,Z 686.096,A -85,B 0,C 180,E1 -7907.396,E2 -7907.396} C_VEL
LIN {X 0,Y 461.269,Z 697.172,A -85,B 0,C 180,E1 -7908.464,E2 -7908.464} C_VEL
LIN {X 0,Y 460.939,Z 705.543,A -85,B 0,C 180,E1 -7909.457,E2 -7909.457} C_VEL
LIN {X 0,Y 460.535,Z 714.614,A -85,B 0,C 180,E1 -7910.779,E2 -7910.779} C_VEL
LIN {X 0,Y 460.171,Z 721.903,A -85,B 0,C 180,E1 -7912.099,E2 -7912.099} C_VEL
LIN {X 0,Y 459.939,Z 727.363,A -85,B 0,C 180,E1 -7913.328,E2 -7913.328} C_VEL
LIN {X 0,Y 459.747,Z 732.299,A -85,B 0,C 180,E1 -7914.737,E2 -7914.737} C_VEL
LIN {X 0,Y 459.748,Z 734.686,A -85,B 0,C 180,E1 -7915.616,E2 -7915.616} C_VEL
LIN {X 0,Y 459.72,Z 736.645,A -85,B 0,C 180,E1 -7916.494,E2 -7916.494} C_VEL
LIN {X 0,Y 459.647,Z 738.178,A -85,B 0,C 180,E1 -7917.371,E2 -7917.371} C_VEL
LIN {X 0,Y 459.604,Z 739.242,A -85,B 0,C 180,E1 -7918.247,E2 -7918.247} C_VEL
LIN {X 0,Y 459.555,Z 739.916,A -85,B 0,C 180,E1 -7919.124,E2 -7919.124} C_VEL
LIN {X 0,Y 459.531,Z 740.196,A -85,B 0,C 180,E1 -7920,E2 -7920} C_VEL
LIN {X 0,Y 459.555,Z 740.027,A -85,B 0,C 180,E1 -7920.876,E2 -7920.876} C_VEL
LIN {X 0,Y 459.635,Z 739.444,A -85,B 0,C 180,E1 -7921.752,E2 -7921.752} C_VEL
LIN {X 0,Y 459.657,Z 738.469,A -85,B 0,C 180,E1 -7922.629,E2 -7922.629} C_VEL
LIN {X 0,Y 459.722,Z 737.061,A -85,B 0,C 180,E1 -7923.506,E2 -7923.506} C_VEL
LIN {X 0,Y 459.731,Z 734.114,A -85,B 0,C 180,E1 -7924.823,E2 -7924.823} C_VEL
LIN {X 0,Y 460.029,Z 728.92,A -85,B 0,C 180,E1 -7926.459,E2 -7926.459} C_VEL
LIN {X 0,Y 460.194,Z 722.852,A -85,B 0,C 180,E1 -7927.9,E2 -7927.9} C_VEL
LIN {X 0,Y 460.53,Z 715.745,A -85,B 0,C 180,E1 -7929.221,E2 -7929.221} C_VEL
LIN {X 0,Y 460.943,Z 706.909,A -85,B 0,C 180,E1 -7930.542,E2 -7930.542} C_VEL
LIN {X 0,Y 461.407,Z 696.694,A -85,B 0,C 180,E1 -7931.755,E2 -7931.755} C_VEL
LIN {X 0,Y 461.891,Z 686.978,A -85,B 0,C 180,E1 -7932.687,E2 -7932.687} C_VEL
LIN {X 0,Y 462.289,Z 676.505,A -85,B 0,C 180,E1 -7933.506,E2 -7933.506} C_VEL
LIN {X 0,Y 462.63,Z 664.573,A -85,B 0,C 180,E1 -7934.236,E2 -7934.236} C_VEL
LIN {X 0,Y 463.099,Z 651.264,A -85,B 0,C 180,E1 -7934.838,E2 -7934.838} C_VEL
LIN {X 0,Y 463.388,Z 637.516,A -85,B 0,C 180,E1 -7935.251,E2 -7935.251} C_VEL
LIN {X 0,Y 464.598,Z 540.811,A -85,B 0,C 180,E1 -7937.024,E2 -7937.024} C_VEL
LIN {X 0,Y 462.489,Z 528.925,A -85,B 0,C 180,E1 -7937.36,E2 -7937.36} C_VEL
LIN {X 0,Y 463.058,Z 510.161,A -85,B 0,C 180,E1 -7940.208,E2 -7940.208} C_VEL
LIN {X 0,Y 463.667,Z 488.619,A -85,B 0,C 180,E1 -7943.446,E2 -7943.446} C_VEL
LIN {X 0,Y 463.797,Z 479.616,A -85,B 0,C 180,E1 -7944.776,E2 -7944.776} C_VEL
LIN {X 0,Y 461.775,Z 469.407,A -85,B 0,C 180,E1 -7946.434,E2 -7946.434} C_VEL
LIN {X 0,Y 460.651,Z 464.731,A -85,B 0,C 180,E1 -7947.208,E2 -7947.208} C_VEL
LIN {X 0,Y 460.516,Z 464.752,A -85,B 0,C 180,E1 -7950.24,E2 -7950.24} C_VEL
LIN {X 0,Y 460.534,Z 464.744,A -85,B 0,C 180,E1 -7953.324,E2 -7953.324} C_VEL
LIN {X 0,Y 460.484,Z 464.751,A -85,B 0,C 180,E1 -7956.529,E2 -7956.529} C_VEL
LIN {X 0,Y 460.562,Z 464.743,A -85,B 0,C 180,E1 -7959.859,E2 -7959.859} C_VEL
LIN {X 0,Y 460.517,Z 464.745,A -85,B 0,C 180,E1 -7962.9,E2 -7962.9} C_VEL
LIN {X 0,Y 460.513,Z 464.748,A -85,B 0,C 180,E1 -7965.83,E2 -7965.83} C_VEL
LIN {X 0,Y 460.535,Z 464.741,A -85,B 0,C 180,E1 -7968.988,E2 -7968.988} C_VEL
LIN {X 0,Y 460.523,Z 464.744,A -85,B 0,C 180,E1 -7971.266,E2 -7971.266} C_VEL
LIN {X 0,Y 460.515,Z 464.745,A -85,B 0,C 180,E1 -7974.554,E2 -7974.554} C_VEL
LIN {X 0,Y 460.536,Z 464.747,A -85,B 0,C 180,E1 -7977.715,E2 -7977.715} C_VEL
LIN {X 0,Y 460.573,Z 464.822,A -85,B 0,C 180,E1 -7980.896,E2 -7980.896} C_VEL
LIN {X 0,Y 464.238,Z 479.509,A -85,B 0,C 180,E1 -7983.277,E2 -7983.277} C_VEL
LIN {X 0,Y 465.507,Z 485.953,A -85,B 0,C 180,E1 -7984.274,E2 -7984.274} C_VEL
LIN {X 0,Y 464.086,Z 507.827,A -85,B 0,C 180,E1 -7987.286,E2 -7987.286} C_VEL
LIN {X 0,Y 463.26,Z 523.052,A -85,B 0,C 180,E1 -7989.369,E2 -7989.369} C_VEL
LIN {X 0,Y 466.122,Z 542.894,A -85,B 0,C 180,E1 -7989.822,E2 -7989.822} C_VEL
LIN {X 0,Y 464.632,Z 659.244,A -85,B 0,C 180,E1 -7991.764,E2 -7991.764} C_VEL
LIN {X 0,Y 464.208,Z 673.546,A -85,B 0,C 180,E1 -7992.174,E2 -7992.174} C_VEL
LIN {X 0,Y 463.692,Z 686.813,A -85,B 0,C 180,E1 -7992.72,E2 -7992.72} C_VEL
LIN {X 0,Y 463.128,Z 700.446,A -85,B 0,C 180,E1 -7993.468,E2 -7993.468} C_VEL
LIN {X 0,Y 462.517,Z 713.124,A -85,B 0,C 180,E1 -7994.352,E2 -7994.352} C_VEL
LIN {X 0,Y 461.844,Z 724.715,A -85,B 0,C 180,E1 -7995.345,E2 -7995.345} C_VEL
LIN {X 0,Y 461.229,Z 736.368,A -85,B 0,C 180,E1 -7996.562,E2 -7996.562} C_VEL
LIN {X 0,Y 460.779,Z 746.758,A -85,B 0,C 180,E1 -7997.893,E2 -7997.893} C_VEL
LIN {X 0,Y 460.326,Z 755.365,A -85,B 0,C 180,E1 -7999.22,E2 -7999.22} C_VEL
LIN {X 0,Y 459.994,Z 763.587,A -85,B 0,C 180,E1 -8000.767,E2 -8000.767} C_VEL
LIN {X 0,Y 459.797,Z 769.355,A -85,B 0,C 180,E1 -8002.092,E2 -8002.092} C_VEL
LIN {X 0,Y 459.713,Z 774.55,A -85,B 0,C 180,E1 -8003.569,E2 -8003.569} C_VEL
LIN {X 0,Y 459.692,Z 777.784,A -85,B 0,C 180,E1 -8004.736,E2 -8004.736} C_VEL
LIN {X 0,Y 459.649,Z 781.403,A -85,B 0,C 180,E1 -8006.493,E2 -8006.493} C_VEL
LIN {X 0,Y 459.629,Z 783.55,A -85,B 0,C 180,E1 -8008.246,E2 -8008.246} C_VEL
LIN {X 0,Y 459.528,Z 784.263,A -85,B 0,C 180,E1 -8009.999,E2 -8009.999} C_VEL
LIN {X 0,Y 459.629,Z 783.554,A -85,B 0,C 180,E1 -8011.751,E2 -8011.751} C_VEL
LIN {X 0,Y 459.648,Z 781.411,A -85,B 0,C 180,E1 -8013.505,E2 -8013.505} C_VEL
LIN {X 0,Y 459.692,Z 777.793,A -85,B 0,C 180,E1 -8015.262,E2 -8015.262} C_VEL
LIN {X 0,Y 459.73,Z 772.595,A -85,B 0,C 180,E1 -8017.024,E2 -8017.024} C_VEL
LIN {X 0,Y 459.842,Z 767.555,A -85,B 0,C 180,E1 -8018.347,E2 -8018.347} C_VEL
LIN {X 0,Y 460.11,Z 760.282,A -85,B 0,C 180,E1 -8019.894,E2 -8019.894} C_VEL
LIN {X 0,Y 460.459,Z 752.666,A -85,B 0,C 180,E1 -8021.22,E2 -8021.22} C_VEL
LIN {X 0,Y 460.868,Z 743.221,A -85,B 0,C 180,E1 -8022.586,E2 -8022.586} C_VEL
LIN {X 0,Y 461.452,Z 732.398,A -85,B 0,C 180,E1 -8023.878,E2 -8023.878} C_VEL
LIN {X 0,Y 462.028,Z 721.142,A -85,B 0,C 180,E1 -8024.985,E2 -8024.985} C_VEL
LIN {X 0,Y 462.674,Z 708.755,A -85,B 0,C 180,E1 -8025.98,E2 -8025.98} C_VEL
LIN {X 0,Y 463.332,Z 694.94,A -85,B 0,C 180,E1 -8026.858,E2 -8026.858} C_VEL
LIN {X 0,Y 463.961,Z 680.519,A -85,B 0,C 180,E1 -8027.557,E2 -8027.557} C_VEL
LIN {X 0,Y 464.443,Z 665.81,A -85,B 0,C 180,E1 -8028.07,E2 -8028.07} C_VEL
LIN {X 0,Y 464.826,Z 650.609,A -85,B 0,C 180,E1 -8028.397,E2 -8028.397} C_VEL
LIN {X 0,Y 465.982,Z 541.144,A -85,B 0,C 180,E1 -8030.21,E2 -8030.21} C_VEL
LIN {X 0,Y 463.245,Z 522.682,A -85,B 0,C 180,E1 -8030.656,E2 -8030.656} C_VEL
LIN {X 0,Y 464.616,Z 499.402,A -85,B 0,C 180,E1 -8033.867,E2 -8033.867} C_VEL
LIN {X 0,Y 465.493,Z 485.942,A -85,B 0,C 180,E1 -8035.724,E2 -8035.724} C_VEL
LIN {X 0,Y 463.351,Z 475.812,A -85,B 0,C 180,E1 -8037.308,E2 -8037.308} C_VEL
LIN {X 0,Y 460.551,Z 464.741,A -85,B 0,C 180,E1 -8039.135,E2 -8039.135} C_VEL
LIN {X 0,Y 460.528,Z 464.747,A -85,B 0,C 180,E1 -8042.283,E2 -8042.283} C_VEL
LIN {X 0,Y 460.508,Z 464.736,A -85,B 0,C 180,E1 -8045.444,E2 -8045.444} C_VEL
LIN {X 0,Y 460.563,Z 464.74,A -85,B 0,C 180,E1 -8048.9,E2 -8048.9} C_VEL
LIN {X 0,Y 460.541,Z 464.742,A -85,B 0,C 180,E1 -8052.177,E2 -8052.177} C_VEL
LIN {X 0,Y 460.514,Z 464.742,A -85,B 0,C 180,E1 -8055.411,E2 -8055.411} C_VEL
LIN {X 0,Y 460.536,Z 464.741,A -85,B 0,C 180,E1 -8058.395,E2 -8058.395} C_VEL
LIN {X 0,Y 460.538,Z 464.739,A -85,B 0,C 180,E1 -8061.268,E2 -8061.268} C_VEL
LIN {X 0,Y 460.504,Z 464.735,A -85,B 0,C 180,E1 -8064.554,E2 -8064.554} C_VEL
LIN {X 0,Y 460.523,Z 464.74,A -85,B 0,C 180,E1 -8067.715,E2 -8067.715} C_VEL
LIN {X 0,Y 460.538,Z 464.744,A -85,B 0,C 180,E1 -8070.769,E2 -8070.769} C_VEL
LIN {X 0,Y 460.557,Z 464.737,A -85,B 0,C 180,E1 -8073.734,E2 -8073.734} C_VEL
LIN {X 0,Y 460.535,Z 464.733,A -85,B 0,C 180,E1 -8076.623,E2 -8076.623} C_VEL
LIN {X 0,Y 460.541,Z 464.733,A -85,B 0,C 180,E1 -8079.452,E2 -8079.452} C_VEL
LIN {X 0,Y 460.548,Z 464.741,A -85,B 0,C 180,E1 -8082.23,E2 -8082.23} C_VEL
LIN {X 0,Y 460.554,Z 464.74,A -85,B 0,C 180,E1 -8084.965,E2 -8084.965} C_VEL
LIN {X 0,Y 460.646,Z 464.725,A -85,B 0,C 180,E1 -8087.667,E2 -8087.667} C_VEL
LIN {X 0,Y 460.619,Z 464.731,A -85,B 0,C 180,E1 -8091.224,E2 -8091.224} C_VEL
LIN {X 0,Y 460.702,Z 464.713,A -85,B 0,C 180,E1 -8093.87,E2 -8093.87} C_VEL
LIN {X 0,Y 460.816,Z 464.703,A -85,B 0,C 180,E1 -8097.378,E2 -8097.378} C_VEL
LIN {X 0,Y 460.842,Z 464.701,A -85,B 0,C 180,E1 -8100,E2 -8100} C_VEL
LIN {X 0,Y 460.815,Z 464.706,A -85,B 0,C 180,E1 -8102.623,E2 -8102.623} C_VEL
LIN {X 0,Y 460.699,Z 464.722,A -85,B 0,C 180,E1 -8106.13,E2 -8106.13} C_VEL
LIN {X 0,Y 460.619,Z 464.731,A -85,B 0,C 180,E1 -8108.776,E2 -8108.776} C_VEL
LIN {X 0,Y 460.623,Z 464.732,A -85,B 0,C 180,E1 -8112.457,E2 -8112.457} C_VEL
LIN {X 0,Y 460.611,Z 464.732,A -85,B 0,C 180,E1 -8116.008,E2 -8116.008} C_VEL
LIN {X 0,Y 460.559,Z 464.737,A -85,B 0,C 180,E1 -8119.616,E2 -8119.616} C_VEL
LIN {X 0,Y 460.501,Z 464.746,A -85,B 0,C 180,E1 -8122.429,E2 -8122.429} C_VEL
LIN {X 0,Y 460.559,Z 464.736,A -85,B 0,C 180,E1 -8125.803,E2 -8125.803} C_VEL
LIN {X 0,Y 460.549,Z 464.742,A -85,B 0,C 180,E1 -8128.233,E2 -8128.233} C_VEL
LIN {X 0,Y 460.516,Z 464.742,A -85,B 0,C 180,E1 -8131.285,E2 -8131.285} C_VEL
LIN {X 0,Y 460.526,Z 464.745,A -85,B 0,C 180,E1 -8134.507,E2 -8134.507} C_VEL
LIN {X 0,Y 460.523,Z 464.74,A -85,B 0,C 180,E1 -8137.621,E2 -8137.621} C_VEL
LIN {X 0,Y 460.552,Z 464.742,A -85,B 0,C 180,E1 -8140.273,E2 -8140.273} C_VEL
LIN {X 0,Y 460.493,Z 464.745,A -85,B 0,C 180,E1 -8143.377,E2 -8143.377} C_VEL
LIN {X 0,Y 460.519,Z 464.749,A -85,B 0,C 180,E1 -8146.629,E2 -8146.629} C_VEL
LIN {X 0,Y 460.555,Z 464.739,A -85,B 0,C 180,E1 -8149.729,E2 -8149.729} C_VEL
LIN {X 0,Y 460.525,Z 464.741,A -85,B 0,C 180,E1 -8152.52,E2 -8152.52} C_VEL
LIN {X 0,Y 460.545,Z 464.74,A -85,B 0,C 180,E1 -8155.625,E2 -8155.625} C_VEL
LIN {X 0,Y 460.534,Z 464.742,A -85,B 0,C 180,E1 -8158.746,E2 -8158.746} C_VEL
LIN {X 0,Y 460.557,Z 464.744,A -85,B 0,C 180,E1 -8161.769,E2 -8161.769} C_VEL
LIN {X 0,Y 460.633,Z 464.87,A -85,B 0,C 180,E1 -8163.038,E2 -8163.038} C_VEL
LIN {X 0,Y 463.271,Z 477.236,A -85,B 0,C 180,E1 -8165.537,E2 -8165.537} C_VEL
LIN {X 0,Y 463.852,Z 481.314,A -85,B 0,C 180,E1 -8166.329,E2 -8166.329} C_VEL
LIN {X 0,Y 462.829,Z 499.234,A -85,B 0,C 180,E1 -8169.56,E2 -8169.56} C_VEL
LIN {X 0,Y 462.073,Z 515.77,A -85,B 0,C 180,E1 -8172.462,E2 -8172.462} C_VEL
LIN {X 0,Y 465.274,Z 533.187,A -85,B 0,C 180,E1 -8172.875,E2 -8172.875} C_VEL
LIN {X 0,Y 465.216,Z 543.526,A -85,B 0,C 180,E1 -8173.026,E2 -8173.026} C_VEL
LIN {X 0,Y 464.542,Z 549.38,A -85,B 0,C 180,E1 -8173.084,E2 -8173.084} C_VEL
LIN {X 0,Y 459.01,Z 568.429,A -85,B 0,C 180,E1 -8173.132,E2 -8173.132} C_VEL
LIN {X 0,Y 458.378,Z 574.282,A -85,B 0,C 180,E1 -8173.192,E2 -8173.192} C_VEL
LIN {X 0,Y 457.959,Z 626.878,A -85,B 0,C 180,E1 -8173.966,E2 -8173.966} C_VEL
LIN {X 0,Y 457.694,Z 639.834,A -85,B 0,C 180,E1 -8174.328,E2 -8174.328} C_VEL
LIN {X 0,Y 457.22,Z 652.327,A -85,B 0,C 180,E1 -8174.854,E2 -8174.854} C_VEL
LIN {X 0,Y 456.74,Z 663.91,A -85,B 0,C 180,E1 -8175.521,E2 -8175.521} C_VEL
LIN {X 0,Y 456.129,Z 674.853,A -85,B 0,C 180,E1 -8176.334,E2 -8176.334} C_VEL
LIN {X 0,Y 455.471,Z 685.152,A -85,B 0,C 180,E1 -8177.299,E2 -8177.299} C_VEL
LIN {X 0,Y 454.892,Z 694.748,A -85,B 0,C 180,E1 -8178.415,E2 -8178.415} C_VEL
LIN {X 0,Y 454.232,Z 704.054,A -85,B 0,C 180,E1 -8179.752,E2 -8179.752} C_VEL
LIN {X 0,Y 453.683,Z 711.472,A -85,B 0,C 180,E1 -8181.09,E2 -8181.09} C_VEL
LIN {X 0,Y 453.27,Z 717.439,A -85,B 0,C 180,E1 -8182.428,E2 -8182.428} C_VEL
LIN {X 0,Y 452.999,Z 722.192,A -85,B 0,C 180,E1 -8183.767,E2 -8183.767} C_VEL
LIN {X 0,Y 452.793,Z 725.886,A -85,B 0,C 180,E1 -8185.104,E2 -8185.104} C_VEL
LIN {X 0,Y 452.718,Z 728.615,A -85,B 0,C 180,E1 -8186.441,E2 -8186.441} C_VEL
LIN {X 0,Y 452.579,Z 730.845,A -85,B 0,C 180,E1 -8188.221,E2 -8188.221} C_VEL
LIN {X 0,Y 452.468,Z 731.636,A -85,B 0,C 180,E1 -8190.001,E2 -8190.001} C_VEL
LIN {X 0,Y 452.58,Z 730.918,A -85,B 0,C 180,E1 -8191.781,E2 -8191.781} C_VEL
LIN {X 0,Y 452.704,Z 728.75,A -85,B 0,C 180,E1 -8193.561,E2 -8193.561} C_VEL
LIN {X 0,Y 452.771,Z 726.087,A -85,B 0,C 180,E1 -8194.899,E2 -8194.899} C_VEL
LIN {X 0,Y 452.998,Z 722.464,A -85,B 0,C 180,E1 -8196.236,E2 -8196.236} C_VEL
LIN {X 0,Y 453.271,Z 717.784,A -85,B 0,C 180,E1 -8197.574,E2 -8197.574} C_VEL
LIN {X 0,Y 453.669,Z 711.897,A -85,B 0,C 180,E1 -8198.913,E2 -8198.913} C_VEL
LIN {X 0,Y 454.144,Z 704.592,A -85,B 0,C 180,E1 -8200.252,E2 -8200.252} C_VEL
LIN {X 0,Y 454.669,Z 697.128,A -85,B 0,C 180,E1 -8201.367,E2 -8201.367} C_VEL
LIN {X 0,Y 455.291,Z 688.071,A -85,B 0,C 180,E1 -8202.482,E2 -8202.482} C_VEL
LIN {X 0,Y 456.032,Z 677.343,A -85,B 0,C 180,E1 -8203.538,E2 -8203.538} C_VEL
LIN {X 0,Y 456.566,Z 666.795,A -85,B 0,C 180,E1 -8204.373,E2 -8204.373} C_VEL
LIN {X 0,Y 457.158,Z 655.125,A -85,B 0,C 180,E1 -8205.094,E2 -8205.094} C_VEL
LIN {X 0,Y 457.605,Z 642.281,A -85,B 0,C 180,E1 -8205.678,E2 -8205.678} C_VEL
LIN {X 0,Y 457.977,Z 629.423,A -85,B 0,C 180,E1 -8206.065,E2 -8206.065} C_VEL
LIN {X 0,Y 458.151,Z 608.921,A -85,B 0,C 180,E1 -8206.402,E2 -8206.402} C_VEL
LIN {X 0,Y 458.484,Z 533.07,A -85,B 0,C 180,E1 -8207.506,E2 -8207.506} C_VEL
LIN {X 0,Y 455.195,Z 515.774,A -85,B 0,C 180,E1 -8207.942,E2 -8207.942} C_VEL
LIN {X 0,Y 456.178,Z 497.338,A -85,B 0,C 180,E1 -8211.227,E2 -8211.227} C_VEL
LIN {X 0,Y 456.919,Z 481.941,A -85,B 0,C 180,E1 -8214.055,E2 -8214.055} C_VEL
LIN {X 0,Y 454.711,Z 470.837,A -85,B 0,C 180,E1 -8216.305,E2 -8216.305} C_VEL
LIN {X 0,Y 453.556,Z 465.62,A -85,B 0,C 180,E1 -8217.389,E2 -8217.389} C_VEL
LIN {X 0,Y 453.483,Z 465.627,A -85,B 0,C 180,E1 -8220.76,E2 -8220.76} C_VEL
LIN {X 0,Y 453.483,Z 465.623,A -85,B 0,C 180,E1 -8223.913,E2 -8223.913} C_VEL
LIN {X 0,Y 453.475,Z 465.622,A -85,B 0,C 180,E1 -8227.189,E2 -8227.189} C_VEL
LIN {X 0,Y 453.523,Z 465.617,A -85,B 0,C 180,E1 -8229.447,E2 -8229.447} C_VEL
LIN {X 0,Y 453.474,Z 465.622,A -85,B 0,C 180,E1 -8232.995,E2 -8232.995} C_VEL
LIN {X 0,Y 453.472,Z 465.627,A -85,B 0,C 180,E1 -8235.779,E2 -8235.779} C_VEL
LIN {X 0,Y 453.485,Z 465.619,A -85,B 0,C 180,E1 -8238.21,E2 -8238.21} C_VEL
LIN {X 0,Y 453.493,Z 465.617,A -85,B 0,C 180,E1 -8240.795,E2 -8240.795} C_VEL
LIN {X 0,Y 453.463,Z 465.626,A -85,B 0,C 180,E1 -8243.918,E2 -8243.918} C_VEL
LIN {X 0,Y 453.489,Z 465.62,A -85,B 0,C 180,E1 -8247.151,E2 -8247.151} C_VEL
LIN {X 0,Y 453.481,Z 465.623,A -85,B 0,C 180,E1 -8250.268,E2 -8250.268} C_VEL
LIN {X 0,Y 453.623,Z 465.763,A -85,B 0,C 180,E1 -8252.71,E2 -8252.71} C_VEL
LIN {X 0,Y 456.66,Z 480.598,A -85,B 0,C 180,E1 -8255.233,E2 -8255.233} C_VEL
LIN {X 0,Y 456.521,Z 489.564,A -85,B 0,C 180,E1 -8256.646,E2 -8256.646} C_VEL
LIN {X 0,Y 455.775,Z 510.535,A -85,B 0,C 180,E1 -8259.934,E2 -8259.934} C_VEL
LIN {X 0,Y 455.211,Z 527.466,A -85,B 0,C 180,E1 -8262.582,E2 -8262.582} C_VEL
LIN {X 0,Y 457.594,Z 542.83,A -85,B 0,C 180,E1 -8262.97,E2 -8262.97} C_VEL
LIN {X 0,Y 456.375,Z 637.313,A -85,B 0,C 180,E1 -8264.652,E2 -8264.652} C_VEL
LIN {X 0,Y 456.137,Z 650.177,A -85,B 0,C 180,E1 -8265.044,E2 -8265.044} C_VEL
LIN {X 0,Y 455.739,Z 662.601,A -85,B 0,C 180,E1 -8265.601,E2 -8265.601} C_VEL
LIN {X 0,Y 455.27,Z 675.555,A -85,B 0,C 180,E1 -8266.384,E2 -8266.384} C_VEL
LIN {X 0,Y 454.896,Z 686.347,A -85,B 0,C 180,E1 -8267.231,E2 -8267.231} C_VEL
LIN {X 0,Y 454.308,Z 697.162,A -85,B 0,C 180,E1 -8268.285,E2 -8268.285} C_VEL
LIN {X 0,Y 453.924,Z 705.601,A -85,B 0,C 180,E1 -8269.292,E2 -8269.292} C_VEL
LIN {X 0,Y 453.552,Z 713.392,A -85,B 0,C 180,E1 -8270.411,E2 -8270.411} C_VEL
LIN {X 0,Y 453.192,Z 720.969,A -85,B 0,C 180,E1 -8271.752,E2 -8271.752} C_VEL
LIN {X 0,Y 452.875,Z 727.952,A -85,B 0,C 180,E1 -8273.316,E2 -8273.316} C_VEL
LIN {X 0,Y 452.697,Z 732.554,A -85,B 0,C 180,E1 -8274.655,E2 -8274.655} C_VEL
LIN {X 0,Y 452.654,Z 734.964,A -85,B 0,C 180,E1 -8275.547,E2 -8275.547} C_VEL
LIN {X 0,Y 452.657,Z 736.935,A -85,B 0,C 180,E1 -8276.439,E2 -8276.439} C_VEL
LIN {X 0,Y 452.571,Z 738.482,A -85,B 0,C 180,E1 -8277.33,E2 -8277.33} C_VEL
LIN {X 0,Y 452.516,Z 739.561,A -85,B 0,C 180,E1 -8278.22,E2 -8278.22} C_VEL
LIN {X 0,Y 452.491,Z 740.241,A -85,B 0,C 180,E1 -8279.11,E2 -8279.11} C_VEL
LIN {X 0,Y 452.465,Z 740.528,A -85,B 0,C 180,E1 -8280,E2 -8280} C_VEL
LIN {X 0,Y 452.491,Z 740.368,A -85,B 0,C 180,E1 -8280.89,E2 -8280.89} C_VEL
LIN {X 0,Y 452.544,Z 739.792,A -85,B 0,C 180,E1 -8281.78,E2 -8281.78} C_VEL
LIN {X 0,Y 452.58,Z 738.821,A -85,B 0,C 180,E1 -8282.67,E2 -8282.67} C_VEL
LIN {X 0,Y 452.661,Z 737.419,A -85,B 0,C 180,E1 -8283.56,E2 -8283.56} C_VEL
LIN {X 0,Y 452.653,Z 734.48,A -85,B 0,C 180,E1 -8284.899,E2 -8284.899} C_VEL
LIN {X 0,Y 452.952,Z 730.45,A -85,B 0,C 180,E1 -8286.235,E2 -8286.235} C_VEL
LIN {X 0,Y 453.106,Z 724.237,A -85,B 0,C 180,E1 -8287.8,E2 -8287.8} C_VEL
LIN {X 0,Y 453.479,Z 717.417,A -85,B 0,C 180,E1 -8289.14,E2 -8289.14} C_VEL
LIN {X 0,Y 453.862,Z 708.836,A -85,B 0,C 180,E1 -8290.483,E2 -8290.483} C_VEL
LIN {X 0,Y 454.282,Z 700.028,A -85,B 0,C 180,E1 -8291.602,E2 -8291.602} C_VEL
LIN {X 0,Y 454.834,Z 689.552,A -85,B 0,C 180,E1 -8292.677,E2 -8292.677} C_VEL
LIN {X 0,Y 455.317,Z 678.445,A -85,B 0,C 180,E1 -8293.592,E2 -8293.592} C_VEL
LIN {X 0,Y 455.654,Z 667.896,A -85,B 0,C 180,E1 -8294.287,E2 -8294.287} C_VEL
LIN {X 0,Y 456.127,Z 655.719,A -85,B 0,C 180,E1 -8294.899,E2 -8294.899} C_VEL
LIN {X 0,Y 456.48,Z 642.375,A -85,B 0,C 180,E1 -8295.373,E2 -8295.373} C_VEL
LIN {X 0,Y 456.685,Z 628.269,A -85,B 0,C 180,E1 -8295.68,E2 -8295.68} C_VEL
LIN {X 0,Y 458.019,Z 542.469,A -85,B 0,C 180,E1 -8297.283,E2 -8297.283} C_VEL
LIN {X 0,Y 455.694,Z 529.344,A -85,B 0,C 180,E1 -8297.674,E2 -8297.674} C_VEL
LIN {X 0,Y 456.302,Z 509.219,A -85,B 0,C 180,E1 -8300.747,E2 -8300.747} C_VEL
LIN {X 0,Y 456.859,Z 492.137,A -85,B 0,C 180,E1 -8303.336,E2 -8303.336} C_VEL
LIN {X 0,Y 457.1,Z 481.805,A -85,B 0,C 180,E1 -8304.886,E2 -8304.886} C_VEL
LIN {X 0,Y 455.251,Z 472.291,A -85,B 0,C 180,E1 -8306.441,E2 -8306.441} C_VEL
LIN {X 0,Y 453.566,Z 465.615,A -85,B 0,C 180,E1 -8307.575,E2 -8307.575} C_VEL
LIN {X 0,Y 453.481,Z 465.626,A -85,B 0,C 180,E1 -8310.759,E2 -8310.759} C_VEL
LIN {X 0,Y 453.483,Z 465.625,A -85,B 0,C 180,E1 -8313.912,E2 -8313.912} C_VEL
LIN {X 0,Y 453.475,Z 465.622,A -85,B 0,C 180,E1 -8317.187,E2 -8317.187} C_VEL
LIN {X 0,Y 453.521,Z 465.617,A -85,B 0,C 180,E1 -8319.446,E2 -8319.446} C_VEL
LIN {X 0,Y 453.467,Z 465.623,A -85,B 0,C 180,E1 -8322.994,E2 -8322.994} C_VEL
LIN {X 0,Y 453.468,Z 465.625,A -85,B 0,C 180,E1 -8325.778,E2 -8325.778} C_VEL
LIN {X 0,Y 453.484,Z 465.621,A -85,B 0,C 180,E1 -8328.209,E2 -8328.209} C_VEL
LIN {X 0,Y 453.491,Z 465.617,A -85,B 0,C 180,E1 -8330.794,E2 -8330.794} C_VEL
LIN {X 0,Y 453.458,Z 465.625,A -85,B 0,C 180,E1 -8333.917,E2 -8333.917} C_VEL
LIN {X 0,Y 453.487,Z 465.624,A -85,B 0,C 180,E1 -8337.151,E2 -8337.151} C_VEL
LIN {X 0,Y 453.512,Z 465.736,A -85,B 0,C 180,E1 -8340.557,E2 -8340.557} C_VEL
LIN {X 0,Y 457.319,Z 480.715,A -85,B 0,C 180,E1 -8343.041,E2 -8343.041} C_VEL
LIN {X 0,Y 458.701,Z 487.463,A -85,B 0,C 180,E1 -8344.108,E2 -8344.108} C_VEL
LIN {X 0,Y 457.199,Z 509.427,A -85,B 0,C 180,E1 -8347.184,E2 -8347.184} C_VEL
LIN {X 0,Y 456.388,Z 522.704,A -85,B 0,C 180,E1 -8349.049,E2 -8349.049} C_VEL
LIN {X 0,Y 459.396,Z 543.452,A -85,B 0,C 180,E1 -8349.55,E2 -8349.55} C_VEL
LIN {X 0,Y 457.831,Z 659.126,A -85,B 0,C 180,E1 -8351.512,E2 -8351.512} C_VEL
LIN {X 0,Y 457.401,Z 673.358,A -85,B 0,C 180,E1 -8351.929,E2 -8351.929} C_VEL
LIN {X 0,Y 456.852,Z 686.776,A -85,B 0,C 180,E1 -8352.492,E2 -8352.492} C_VEL
LIN {X 0,Y 456.228,Z 699.741,A -85,B 0,C 180,E1 -8353.211,E2 -8353.211} C_VEL
LIN {X 0,Y 455.605,Z 712.484,A -85,B 0,C 180,E1 -8354.108,E2 -8354.108} C_VEL
LIN {X 0,Y 454.885,Z 724.119,A -85,B 0,C 180,E1 -8355.115,E2 -8355.115} C_VEL
LIN {X 0,Y 454.24,Z 735.815,A -85,B 0,C 180,E1 -8356.351,E2 -8356.351} C_VEL
LIN {X 0,Y 453.751,Z 746.239,A -85,B 0,C 180,E1 -8357.703,E2 -8357.703} C_VEL
LIN {X 0,Y 453.291,Z 754.869,A -85,B 0,C 180,E1 -8359.05,E2 -8359.05} C_VEL
LIN {X 0,Y 452.942,Z 763.112,A -85,B 0,C 180,E1 -8360.622,E2 -8360.622} C_VEL
LIN {X 0,Y 452.721,Z 768.897,A -85,B 0,C 180,E1 -8361.968,E2 -8361.968} C_VEL
LIN {X 0,Y 452.607,Z 774.509,A -85,B 0,C 180,E1 -8363.607,E2 -8363.607} C_VEL
LIN {X 0,Y 452.554,Z 778.419,A -85,B 0,C 180,E1 -8365.099,E2 -8365.099} C_VEL
LIN {X 0,Y 452.547,Z 780.981,A -85,B 0,C 180,E1 -8366.437,E2 -8366.437} C_VEL
LIN {X 0,Y 452.538,Z 783.138,A -85,B 0,C 180,E1 -8368.219,E2 -8368.219} C_VEL
LIN {X 0,Y 452.462,Z 783.856,A -85,B 0,C 180,E1 -8369.999,E2 -8369.999} C_VEL
LIN {X 0,Y 452.538,Z 783.141,A -85,B 0,C 180,E1 -8371.779,E2 -8371.779} C_VEL
LIN {X 0,Y 452.546,Z 780.988,A -85,B 0,C 180,E1 -8373.56,E2 -8373.56} C_VEL
LIN {X 0,Y 452.598,Z 777.358,A -85,B 0,C 180,E1 -8375.345,E2 -8375.345} C_VEL
LIN {X 0,Y 452.65,Z 772.144,A -85,B 0,C 180,E1 -8377.134,E2 -8377.134} C_VEL
LIN {X 0,Y 452.776,Z 767.087,A -85,B 0,C 180,E1 -8378.478,E2 -8378.478} C_VEL
LIN {X 0,Y 453.057,Z 759.795,A -85,B 0,C 180,E1 -8380.049,E2 -8380.049} C_VEL
LIN {X 0,Y 453.421,Z 752.156,A -85,B 0,C 180,E1 -8381.397,E2 -8381.397} C_VEL
LIN {X 0,Y 453.83,Z 743.473,A -85,B 0,C 180,E1 -8382.678,E2 -8382.678} C_VEL
LIN {X 0,Y 454.421,Z 732.834,A -85,B 0,C 180,E1 -8383.983,E2 -8383.983} C_VEL
LIN {X 0,Y 455.031,Z 721.74,A -85,B 0,C 180,E1 -8385.106,E2 -8385.106} C_VEL
LIN {X 0,Y 455.709,Z 709.605,A -85,B 0,C 180,E1 -8386.116,E2 -8386.116} C_VEL
LIN {X 0,Y 456.377,Z 696.103,A -85,B 0,C 180,E1 -8387.012,E2 -8387.012} C_VEL
LIN {X 0,Y 457.049,Z 681.894,A -85,B 0,C 180,E1 -8387.731,E2 -8387.731} C_VEL
LIN {X 0,Y 457.566,Z 667.427,A -85,B 0,C 180,E1 -8388.265,E2 -8388.265} C_VEL
LIN {X 0,Y 457.973,Z 653.643,A -85,B 0,C 180,E1 -8388.595,E2 -8388.595} C_VEL
LIN {X 0,Y 459.29,Z 542.102,A -85,B 0,C 180,E1 -8390.474,E2 -8390.474} C_VEL
LIN {X 0,Y 456.383,Z 522.655,A -85,B 0,C 180,E1 -8390.949,E2 -8390.949} C_VEL
LIN {X 0,Y 457.76,Z 500.886,A -85,B 0,C 180,E1 -8394.006,E2 -8394.006} C_VEL
LIN {X 0,Y 458.689,Z 487.446,A -85,B 0,C 180,E1 -8395.89,E2 -8395.89} C_VEL
LIN {X 0,Y 455.837,Z 474.708,A -85,B 0,C 180,E1 -8397.936,E2 -8397.936} C_VEL
LIN {X 0,Y 453.509,Z 465.618,A -85,B 0,C 180,E1 -8399.472,E2 -8399.472} C_VEL
LIN {X 0,Y 453.478,Z 465.626,A -85,B 0,C 180,E1 -8402.847,E2 -8402.847} C_VEL
LIN {X 0,Y 453.452,Z 465.618,A -85,B 0,C 180,E1 -8406.081,E2 -8406.081} C_VEL
LIN {X 0,Y 453.527,Z 465.615,A -85,B 0,C 180,E1 -8409.444,E2 -8409.444} C_VEL
LIN {X 0,Y 453.485,Z 465.623,A -85,B 0,C 180,E1 -8412.99,E2 -8412.99} C_VEL
LIN {X 0,Y 453.469,Z 465.619,A -85,B 0,C 180,E1 -8415.779,E2 -8415.779} C_VEL
LIN {X 0,Y 453.488,Z 465.618,A -85,B 0,C 180,E1 -8418.21,E2 -8418.21} C_VEL
LIN {X 0,Y 453.524,Z 465.617,A -85,B 0,C 180,E1 -8420.786,E2 -8420.786} C_VEL
LIN {X 0,Y 453.448,Z 465.612,A -85,B 0,C 180,E1 -8423.917,E2 -8423.917} C_VEL
LIN {X 0,Y 453.473,Z 465.62,A -85,B 0,C 180,E1 -8427.15,E2 -8427.15} C_VEL
LIN {X 0,Y 453.504,Z 465.618,A -85,B 0,C 180,E1 -8430.27,E2 -8430.27} C_VEL
LIN {X 0,Y 453.503,Z 465.617,A -85,B 0,C 180,E1 -8433.294,E2 -8433.294} C_VEL
LIN {X 0,Y 453.493,Z 465.617,A -85,B 0,C 180,E1 -8436.238,E2 -8436.238} C_VEL
LIN {X 0,Y 453.472,Z 465.615,A -85,B 0,C 180,E1 -8439.117,E2 -8439.117} C_VEL
LIN {X 0,Y 453.501,Z 465.617,A -85,B 0,C 180,E1 -8441.944,E2 -8441.944} C_VEL
LIN {X 0,Y 453.529,Z 465.615,A -85,B 0,C 180,E1 -8444.726,E2 -8444.726} C_VEL
LIN {X 0,Y 453.59,Z 465.604,A -85,B 0,C 180,E1 -8447.472,E2 -8447.472} C_VEL
LIN {X 0,Y 453.582,Z 465.608,A -85,B 0,C 180,E1 -8451.087,E2 -8451.087} C_VEL
LIN {X 0,Y 453.669,Z 465.589,A -85,B 0,C 180,E1 -8453.775,E2 -8453.775} C_VEL
LIN {X 0,Y 453.756,Z 465.582,A -85,B 0,C 180,E1 -8457.337,E2 -8457.337} C_VEL
LIN {X 0,Y 453.813,Z 465.577,A -85,B 0,C 180,E1 -8460,E2 -8460} C_VEL
LIN {X 0,Y 453.756,Z 465.585,A -85,B 0,C 180,E1 -8462.663,E2 -8462.663} C_VEL
LIN {X 0,Y 453.667,Z 465.599,A -85,B 0,C 180,E1 -8466.226,E2 -8466.226} C_VEL
LIN {X 0,Y 453.582,Z 465.608,A -85,B 0,C 180,E1 -8468.914,E2 -8468.914} C_VEL
LIN {X 0,Y 453.59,Z 465.607,A -85,B 0,C 180,E1 -8472.551,E2 -8472.551} C_VEL
LIN {X 0,Y 453.546,Z 465.614,A -85,B 0,C 180,E1 -8476.196,E2 -8476.196} C_VEL
LIN {X 0,Y 453.51,Z 465.617,A -85,B 0,C 180,E1 -8479.042,E2 -8479.042} C_VEL
LIN {X 0,Y 453.466,Z 465.619,A -85,B 0,C 180,E1 -8481.837,E2 -8481.837} C_VEL
LIN {X 0,Y 453.504,Z 465.62,A -85,B 0,C 180,E1 -8484.735,E2 -8484.735} C_VEL
LIN {X 0,Y 453.529,Z 465.613,A -85,B 0,C 180,E1 -8487.962,E2 -8487.962} C_VEL
LIN {X 0,Y 453.474,Z 465.623,A -85,B 0,C 180,E1 -8490.76,E2 -8490.76} C_VEL
LIN {X 0,Y 453.47,Z 465.619,A -85,B 0,C 180,E1 -8493.914,E2 -8493.914} C_VEL
LIN {X 0,Y 453.464,Z 465.62,A -85,B 0,C 180,E1 -8497.189,E2 -8497.189} C_VEL
LIN {X 0,Y 453.526,Z 465.614,A -85,B 0,C 180,E1 -8499.446,E2 -8499.446} C_VEL
LIN {X 0,Y 453.456,Z 465.624,A -85,B 0,C 180,E1 -8502.996,E2 -8502.996} C_VEL
LIN {X 0,Y 453.471,Z 465.621,A -85,B 0,C 180,E1 -8505.782,E2 -8505.782} C_VEL
LIN {X 0,Y 453.491,Z 465.622,A -85,B 0,C 180,E1 -8508.213,E2 -8508.213} C_VEL
LIN {X 0,Y 453.528,Z 465.618,A -85,B 0,C 180,E1 -8510.789,E2 -8510.789} C_VEL
LIN {X 0,Y 453.453,Z 465.622,A -85,B 0,C 180,E1 -8513.919,E2 -8513.919} C_VEL
LIN {X 0,Y 453.48,Z 465.623,A -85,B 0,C 180,E1 -8517.153,E2 -8517.153} C_VEL
LIN {X 0,Y 453.511,Z 465.62,A -85,B 0,C 180,E1 -8520.273,E2 -8520.273} C_VEL
LIN {X 0,Y 453.597,Z 465.785,A -85,B 0,C 180,E1 -8522.741,E2 -8522.741} C_VEL
LIN {X 0,Y 456.401,Z 478.903,A -85,B 0,C 180,E1 -8525.434,E2 -8525.434} C_VEL
LIN {X 0,Y 456.977,Z 482.739,A -85,B 0,C 180,E1 -8526.191,E2 -8526.191} C_VEL
LIN {X 0,Y 456.006,Z 499.405,A -85,B 0,C 180,E1 -8529.24,E2 -8529.24} C_VEL
LIN {X 0,Y 455.205,Z 516.2,A -85,B 0,C 180,E1 -8532.183,E2 -8532.183} C_VEL
LIN {X 0,Y 458.554,Z 533.948,A -85,B 0,C 180,E1 -8532.6,E2 -8532.6} C_VEL
LIN {X 0,Y 458.378,Z 574.282,A -85,B 0,C 180,E1 -8533.192,E2 -8533.192} C_VEL
LIN {X 0,Y 457.745,Z 580.131,A -85,B 0,C 180,E1 -8533.252,E2 -8533.252} C_VEL
LIN {X 0,Y 452.149,Z 599.16,A -85,B 0,C 180,E1 -8533.298,E2 -8533.298} C_VEL
LIN {X 0,Y 451.426,Z 605.013,A -85,B 0,C 180,E1 -8533.355,E2 -8533.355} C_VEL
LIN {X 0,Y 451.215,Z 628.154,A -85,B 0,C 180,E1 -8533.719,E2 -8533.719} C_VEL
LIN {X 0,Y 450.91,Z 640.768,A -85,B 0,C 180,E1 -8534.086,E2 -8534.086} C_VEL
LIN {X 0,Y 450.415,Z 653.096,A -85,B 0,C 180,E1 -8534.619,E2 -8534.619} C_VEL
LIN {X 0,Y 449.902,Z 664.58,A -85,B 0,C 180,E1 -8535.296,E2 -8535.296} C_VEL
LIN {X 0,Y 449.258,Z 675.59,A -85,B 0,C 180,E1 -8536.135,E2 -8536.135} C_VEL
LIN {X 0,Y 448.577,Z 685.691,A -85,B 0,C 180,E1 -8537.101,E2 -8537.101} C_VEL
LIN {X 0,Y 447.961,Z 695.259,A -85,B 0,C 180,E1 -8538.233,E2 -8538.233} C_VEL
LIN {X 0,Y 447.246,Z 704.538,A -85,B 0,C 180,E1 -8539.59,E2 -8539.59} C_VEL
LIN {X 0,Y 446.7,Z 711.93,A -85,B 0,C 180,E1 -8540.949,E2 -8540.949} C_VEL
LIN {X 0,Y 446.243,Z 717.884,A -85,B 0,C 180,E1 -8542.308,E2 -8542.308} C_VEL
LIN {X 0,Y 445.97,Z 722.624,A -85,B 0,C 180,E1 -8543.668,E2 -8543.668} C_VEL
LIN {X 0,Y 445.726,Z 726.31,A -85,B 0,C 180,E1 -8545.026,E2 -8545.026} C_VEL
LIN {X 0,Y 445.659,Z 729.031,A -85,B 0,C 180,E1 -8546.385,E2 -8546.385} C_VEL
LIN {X 0,Y 445.522,Z 731.254,A -85,B 0,C 180,E1 -8548.193,E2 -8548.193} C_VEL
LIN {X 0,Y 445.404,Z 732.044,A -85,B 0,C 180,E1 -8550.001,E2 -8550.001} C_VEL
LIN {X 0,Y 445.523,Z 731.327,A -85,B 0,C 180,E1 -8551.809,E2 -8551.809} C_VEL
LIN {X 0,Y 445.645,Z 729.164,A -85,B 0,C 180,E1 -8553.618,E2 -8553.618} C_VEL
LIN {X 0,Y 445.689,Z 726.51,A -85,B 0,C 180,E1 -8554.977,E2 -8554.977} C_VEL
LIN {X 0,Y 446.055,Z 721.921,A -85,B 0,C 180,E1 -8556.654,E2 -8556.654} C_VEL
LIN {X 0,Y 446.35,Z 716.421,A -85,B 0,C 180,E1 -8558.148,E2 -8558.148} C_VEL
LIN {X 0,Y 446.934,Z 708.9,A -85,B 0,C 180,E1 -8559.733,E2 -8559.733} C_VEL
LIN {X 0,Y 447.556,Z 700.774,A -85,B 0,C 180,E1 -8561.092,E2 -8561.092} C_VEL
LIN {X 0,Y 448.111,Z 692.423,A -85,B 0,C 180,E1 -8562.225,E2 -8562.225} C_VEL
LIN {X 0,Y 448.87,Z 682.121,A -85,B 0,C 180,E1 -8563.354,E2 -8563.354} C_VEL
LIN {X 0,Y 449.509,Z 671.16,A -85,B 0,C 180,E1 -8564.318,E2 -8564.318} C_VEL
LIN {X 0,Y 450.138,Z 660.677,A -85,B 0,C 180,E1 -8565.045,E2 -8565.045} C_VEL
LIN {X 0,Y 450.645,Z 649.169,A -85,B 0,C 180,E1 -8565.665,E2 -8565.665} C_VEL
LIN {X 0,Y 450.996,Z 636.724,A -85,B 0,C 180,E1 -8566.146,E2 -8566.146} C_VEL
LIN {X 0,Y 451.296,Z 623.927,A -85,B 0,C 180,E1 -8566.454,E2 -8566.454} C_VEL
LIN {X 0,Y 451.759,Z 533.954,A -85,B 0,C 180,E1 -8567.788,E2 -8567.788} C_VEL
LIN {X 0,Y 448.286,Z 515.853,A -85,B 0,C 180,E1 -8568.25,E2 -8568.25} C_VEL
LIN {X 0,Y 449.265,Z 498.79,A -85,B 0,C 180,E1 -8571.329,E2 -8571.329} C_VEL
LIN {X 0,Y 450.055,Z 483.422,A -85,B 0,C 180,E1 -8574.19,E2 -8574.19} C_VEL
LIN {X 0,Y 447.554,Z 471.078,A -85,B 0,C 180,E1 -8576.733,E2 -8576.733} C_VEL
LIN {X 0,Y 446.5,Z 466.5,A -85,B 0,C 180,E1 -8577.732,E2 -8577.732} C_VEL
LIN {X 0,Y 446.422,Z 466.506,A -85,B 0,C 180,E1 -8581.301,E2 -8581.301} C_VEL
LIN {X 0,Y 446.435,Z 466.498,A -85,B 0,C 180,E1 -8584.524,E2 -8584.524} C_VEL
LIN {X 0,Y 446.436,Z 466.498,A -85,B 0,C 180,E1 -8588.082,E2 -8588.082} C_VEL
LIN {X 0,Y 446.434,Z 466.497,A -85,B 0,C 180,E1 -8590.918,E2 -8590.918} C_VEL
LIN {X 0,Y 446.429,Z 466.498,A -85,B 0,C 180,E1 -8593.844,E2 -8593.844} C_VEL
LIN {X 0,Y 446.405,Z 466.501,A -85,B 0,C 180,E1 -8596.404,E2 -8596.404} C_VEL
LIN {X 0,Y 446.432,Z 466.496,A -85,B 0,C 180,E1 -8599.083,E2 -8599.083} C_VEL
LIN {X 0,Y 446.432,Z 466.495,A -85,B 0,C 180,E1 -8602.123,E2 -8602.123} C_VEL
LIN {X 0,Y 446.437,Z 466.502,A -85,B 0,C 180,E1 -8605.477,E2 -8605.477} C_VEL
LIN {X 0,Y 446.422,Z 466.499,A -85,B 0,C 180,E1 -8608.7,E2 -8608.7} C_VEL
LIN {X 0,Y 446.491,Z 466.495,A -85,B 0,C 180,E1 -8611.822,E2 -8611.822} C_VEL
LIN {X 0,Y 446.535,Z 466.56,A -85,B 0,C 180,E1 -8612.462,E2 -8612.462} C_VEL
LIN {X 0,Y 449.67,Z 481.518,A -85,B 0,C 180,E1 -8615.027,E2 -8615.027} C_VEL
LIN {X 0,Y 449.803,Z 486.215,A -85,B 0,C 180,E1 -8615.786,E2 -8615.786} C_VEL
LIN {X 0,Y 449.092,Z 504.424,A -85,B 0,C 180,E1 -8618.663,E2 -8618.663} C_VEL
LIN {X 0,Y 448.367,Z 525.369,A -85,B 0,C 180,E1 -8621.963,E2 -8621.963} C_VEL
LIN {X 0,Y 448.306,Z 527.774,A -85,B 0,C 180,E1 -8622.343,E2 -8622.343} C_VEL
LIN {X 0,Y 450.759,Z 544.043,A -85,B 0,C 180,E1 -8622.75,E2 -8622.75} C_VEL
LIN {X 0,Y 449.454,Z 637.955,A -85,B 0,C 180,E1 -8624.468,E2 -8624.468} C_VEL
LIN {X 0,Y 449.197,Z 650.649,A -85,B 0,C 180,E1 -8624.865,E2 -8624.865} C_VEL
LIN {X 0,Y 448.752,Z 664.064,A -85,B 0,C 180,E1 -8625.488,E2 -8625.488} C_VEL
LIN {X 0,Y 448.289,Z 676.72,A -85,B 0,C 180,E1 -8626.283,E2 -8626.283} C_VEL
LIN {X 0,Y 447.853,Z 687.311,A -85,B 0,C 180,E1 -8627.139,E2 -8627.139} C_VEL
LIN {X 0,Y 447.261,Z 698.055,A -85,B 0,C 180,E1 -8628.213,E2 -8628.213} C_VEL
LIN {X 0,Y 446.844,Z 707.234,A -85,B 0,C 180,E1 -8629.35,E2 -8629.35} C_VEL
LIN {X 0,Y 446.407,Z 716.133,A -85,B 0,C 180,E1 -8630.713,E2 -8630.713} C_VEL
LIN {X 0,Y 446.041,Z 723.292,A -85,B 0,C 180,E1 -8632.075,E2 -8632.075} C_VEL
LIN {X 0,Y 445.798,Z 729.771,A -85,B 0,C 180,E1 -8633.664,E2 -8633.664} C_VEL
LIN {X 0,Y 445.563,Z 734.031,A -85,B 0,C 180,E1 -8635.023,E2 -8635.023} C_VEL
LIN {X 0,Y 445.576,Z 737.194,A -85,B 0,C 180,E1 -8636.383,E2 -8636.383} C_VEL
LIN {X 0,Y 445.499,Z 738.768,A -85,B 0,C 180,E1 -8637.287,E2 -8637.287} C_VEL
LIN {X 0,Y 445.431,Z 739.867,A -85,B 0,C 180,E1 -8638.192,E2 -8638.192} C_VEL
LIN {X 0,Y 445.401,Z 740.863,A -85,B 0,C 180,E1 -8640,E2 -8640} C_VEL
LIN {X 0,Y 445.429,Z 740.72,A -85,B 0,C 180,E1 -8640.904,E2 -8640.904} C_VEL
LIN {X 0,Y 445.457,Z 740.152,A -85,B 0,C 180,E1 -8641.808,E2 -8641.808} C_VEL
LIN {X 0,Y 445.507,Z 739.187,A -85,B 0,C 180,E1 -8642.712,E2 -8642.712} C_VEL
LIN {X 0,Y 445.6,Z 737.793,A -85,B 0,C 180,E1 -8643.617,E2 -8643.617} C_VEL
LIN {X 0,Y 445.582,Z 734.859,A -85,B 0,C 180,E1 -8644.977,E2 -8644.977} C_VEL
LIN {X 0,Y 445.898,Z 730.826,A -85,B 0,C 180,E1 -8646.334,E2 -8646.334} C_VEL
LIN {X 0,Y 446.07,Z 724.603,A -85,B 0,C 180,E1 -8647.924,E2 -8647.924} C_VEL
LIN {X 0,Y 446.481,Z 717.77,A -85,B 0,C 180,E1 -8649.285,E2 -8649.285} C_VEL
LIN {X 0,Y 446.896,Z 709.206,A -85,B 0,C 180,E1 -8650.648,E2 -8650.648} C_VEL
LIN {X 0,Y 447.341,Z 700.427,A -85,B 0,C 180,E1 -8651.785,E2 -8651.785} C_VEL
LIN {X 0,Y 447.915,Z 690.12,A -85,B 0,C 180,E1 -8652.865,E2 -8652.865} C_VEL
LIN {X 0,Y 448.453,Z 678.605,A -85,B 0,C 180,E1 -8653.827,E2 -8653.827} C_VEL
LIN {X 0,Y 448.805,Z 668.37,A -85,B 0,C 180,E1 -8654.51,E2 -8654.51} C_VEL
LIN {X 0,Y 449.3,Z 656.237,A -85,B 0,C 180,E1 -8655.131,E2 -8655.131} C_VEL
LIN {X 0,Y 449.662,Z 642.985,A -85,B 0,C 180,E1 -8655.612,E2 -8655.612} C_VEL
LIN {X 0,Y 449.898,Z 629.087,A -85,B 0,C 180,E1 -8655.923,E2 -8655.923} C_VEL
LIN {X 0,Y 451.344,Z 543.653,A -85,B 0,C 180,E1 -8657.579,E2 -8657.579} C_VEL
LIN {X 0,Y 449.122,Z 530.958,A -85,B 0,C 180,E1 -8657.958,E2 -8657.958} C_VEL
LIN {X 0,Y 448.919,Z 529.698,A -85,B 0,C 180,E1 -8658.013,E2 -8658.013} C_VEL
LIN {X 0,Y 449.522,Z 511.435,A -85,B 0,C 180,E1 -8660.835,E2 -8660.835} C_VEL
LIN {X 0,Y 450.334,Z 489.496,A -85,B 0,C 180,E1 -8664.184,E2 -8664.184} C_VEL
LIN {X 0,Y 450.322,Z 483.14,A -85,B 0,C 180,E1 -8665.15,E2 -8665.15} C_VEL
LIN {X 0,Y 448.197,Z 472.816,A -85,B 0,C 180,E1 -8666.888,E2 -8666.888} C_VEL
LIN {X 0,Y 446.502,Z 466.496,A -85,B 0,C 180,E1 -8668.005,E2 -8668.005} C_VEL
LIN {X 0,Y 446.421,Z 466.505,A -85,B 0,C 180,E1 -8671.3,E2 -8671.3} C_VEL
LIN {X 0,Y 446.436,Z 466.501,A -85,B 0,C 180,E1 -8674.522,E2 -8674.522} C_VEL
LIN {X 0,Y 446.435,Z 466.503,A -85,B 0,C 180,E1 -8678.081,E2 -8678.081} C_VEL
LIN {X 0,Y 446.431,Z 466.5,A -85,B 0,C 180,E1 -8680.917,E2 -8680.917} C_VEL
LIN {X 0,Y 446.404,Z 466.505,A -85,B 0,C 180,E1 -8683.846,E2 -8683.846} C_VEL
LIN {X 0,Y 446.403,Z 466.504,A -85,B 0,C 180,E1 -8686.403,E2 -8686.403} C_VEL
LIN {X 0,Y 446.431,Z 466.498,A -85,B 0,C 180,E1 -8689.082,E2 -8689.082} C_VEL
LIN {X 0,Y 446.412,Z 466.501,A -85,B 0,C 180,E1 -8692.12,E2 -8692.12} C_VEL
LIN {X 0,Y 446.433,Z 466.502,A -85,B 0,C 180,E1 -8695.476,E2 -8695.476} C_VEL
LIN {X 0,Y 446.42,Z 466.503,A -85,B 0,C 180,E1 -8698.699,E2 -8698.699} C_VEL
LIN {X 0,Y 446.467,Z 466.629,A -85,B 0,C 180,E1 -8700.205,E2 -8700.205} C_VEL
LIN {X 0,Y 450.379,Z 481.979,A -85,B 0,C 180,E1 -8702.806,E2 -8702.806} C_VEL
LIN {X 0,Y 451.857,Z 488.967,A -85,B 0,C 180,E1 -8703.934,E2 -8703.934} C_VEL
LIN {X 0,Y 450.454,Z 509.045,A -85,B 0,C 180,E1 -8706.798,E2 -8706.798} C_VEL
LIN {X 0,Y 449.555,Z 522.673,A -85,B 0,C 180,E1 -8708.745,E2 -8708.745} C_VEL
LIN {X 0,Y 452.673,Z 544.427,A -85,B 0,C 180,E1 -8709.276,E2 -8709.276} C_VEL
LIN {X 0,Y 451.057,Z 659.05,A -85,B 0,C 180,E1 -8711.254,E2 -8711.254} C_VEL
LIN {X 0,Y 450.61,Z 673.205,A -85,B 0,C 180,E1 -8711.676,E2 -8711.676} C_VEL
LIN {X 0,Y 450.043,Z 685.738,A -85,B 0,C 180,E1 -8712.204,E2 -8712.204} C_VEL
LIN {X 0,Y 449.383,Z 699.064,A -85,B 0,C 180,E1 -8712.947,E2 -8712.947} C_VEL
LIN {X 0,Y 448.684,Z 711.864,A -85,B 0,C 180,E1 -8713.856,E2 -8713.856} C_VEL
LIN {X 0,Y 447.947,Z 723.545,A -85,B 0,C 180,E1 -8714.879,E2 -8714.879} C_VEL
LIN {X 0,Y 447.269,Z 735.276,A -85,B 0,C 180,E1 -8716.134,E2 -8716.134} C_VEL
LIN {X 0,Y 446.714,Z 745.285,A -85,B 0,C 180,E1 -8717.439,E2 -8717.439} C_VEL
LIN {X 0,Y 446.264,Z 754.388,A -85,B 0,C 180,E1 -8718.876,E2 -8718.876} C_VEL
LIN {X 0,Y 445.897,Z 762.649,A -85,B 0,C 180,E1 -8720.473,E2 -8720.473} C_VEL
LIN {X 0,Y 445.64,Z 768.448,A -85,B 0,C 180,E1 -8721.839,E2 -8721.839} C_VEL
LIN {X 0,Y 445.529,Z 774.385,A -85,B 0,C 180,E1 -8723.613,E2 -8723.613} C_VEL
LIN {X 0,Y 445.487,Z 777.995,A -85,B 0,C 180,E1 -8725.021,E2 -8725.021} C_VEL
LIN {X 0,Y 445.446,Z 780.561,A -85,B 0,C 180,E1 -8726.381,E2 -8726.381} C_VEL
LIN {X 0,Y 445.482,Z 781.827,A -85,B 0,C 180,E1 -8727.286,E2 -8727.286} C_VEL
LIN {X 0,Y 445.425,Z 783.268,A -85,B 0,C 180,E1 -8729.095,E2 -8729.095} C_VEL
LIN {X 0,Y 445.423,Z 783.269,A -85,B 0,C 180,E1 -8730.903,E2 -8730.903} C_VEL
LIN {X 0,Y 445.482,Z 781.832,A -85,B 0,C 180,E1 -8732.712,E2 -8732.712} C_VEL
LIN {X 0,Y 445.421,Z 778.935,A -85,B 0,C 180,E1 -8734.524,E2 -8734.524} C_VEL
LIN {X 0,Y 445.487,Z 775.3,A -85,B 0,C 180,E1 -8736.065,E2 -8736.065} C_VEL
LIN {X 0,Y 445.578,Z 770.13,A -85,B 0,C 180,E1 -8737.703,E2 -8737.703} C_VEL
LIN {X 0,Y 445.822,Z 763.698,A -85,B 0,C 180,E1 -8739.297,E2 -8739.297} C_VEL
LIN {X 0,Y 446.184,Z 755.667,A -85,B 0,C 180,E1 -8740.894,E2 -8740.894} C_VEL
LIN {X 0,Y 446.602,Z 746.442,A -85,B 0,C 180,E1 -8742.389,E2 -8742.389} C_VEL
LIN {X 0,Y 447.152,Z 737.143,A -85,B 0,C 180,E1 -8743.635,E2 -8743.635} C_VEL
LIN {X 0,Y 447.873,Z 725.897,A -85,B 0,C 180,E1 -8744.888,E2 -8744.888} C_VEL
LIN {X 0,Y 448.54,Z 714.725,A -85,B 0,C 180,E1 -8745.913,E2 -8745.913} C_VEL
LIN {X 0,Y 449.19,Z 702.618,A -85,B 0,C 180,E1 -8746.824,E2 -8746.824} C_VEL
LIN {X 0,Y 449.901,Z 689.47,A -85,B 0,C 180,E1 -8747.605,E2 -8747.605} C_VEL
LIN {X 0,Y 450.464,Z 675.451,A -85,B 0,C 180,E1 -8748.239,E2 -8748.239} C_VEL
LIN {X 0,Y 450.992,Z 661.26,A -85,B 0,C 180,E1 -8748.688,E2 -8748.688} C_VEL
LIN {X 0,Y 451.356,Z 640.529,A -85,B 0,C 180,E1 -8749.085,E2 -8749.085} C_VEL
LIN {X 0,Y 452.614,Z 543.586,A -85,B 0,C 180,E1 -8750.736,E2 -8750.736} C_VEL
LIN {X 0,Y 449.545,Z 522.629,A -85,B 0,C 180,E1 -8751.253,E2 -8751.253} C_VEL
LIN {X 0,Y 451.021,Z 500.685,A -85,B 0,C 180,E1 -8754.388,E2 -8754.388} C_VEL
LIN {X 0,Y 451.84,Z 488.941,A -85,B 0,C 180,E1 -8756.064,E2 -8756.064} C_VEL
LIN {X 0,Y 448.608,Z 474.873,A -85,B 0,C 180,E1 -8758.376,E2 -8758.376} C_VEL
LIN {X 0,Y 446.449,Z 466.497,A -85,B 0,C 180,E1 -8759.825,E2 -8759.825} C_VEL
LIN {X 0,Y 446.439,Z 466.498,A -85,B 0,C 180,E1 -8763.452,E2 -8763.452} C_VEL
LIN {X 0,Y 446.404,Z 466.504,A -85,B 0,C 180,E1 -8766.743,E2 -8766.743} C_VEL
LIN {X 0,Y 446.486,Z 466.492,A -85,B 0,C 180,E1 -8769.53,E2 -8769.53} C_VEL
LIN {X 0,Y 446.443,Z 466.501,A -85,B 0,C 180,E1 -8772.601,E2 -8772.601} C_VEL
LIN {X 0,Y 446.45,Z 466.496,A -85,B 0,C 180,E1 -8775.102,E2 -8775.102} C_VEL
LIN {X 0,Y 446.436,Z 466.5,A -85,B 0,C 180,E1 -8778.61,E2 -8778.61} C_VEL
LIN {X 0,Y 446.467,Z 466.494,A -85,B 0,C 180,E1 -8780.975,E2 -8780.975} C_VEL
LIN {X 0,Y 446.412,Z 466.488,A -85,B 0,C 180,E1 -8784.373,E2 -8784.373} C_VEL
LIN {X 0,Y 446.419,Z 466.497,A -85,B 0,C 180,E1 -8787.638,E2 -8787.638} C_VEL
LIN {X 0,Y 446.459,Z 466.498,A -85,B 0,C 180,E1 -8790.791,E2 -8790.791} C_VEL
LIN {X 0,Y 446.467,Z 466.493,A -85,B 0,C 180,E1 -8793.848,E2 -8793.848} C_VEL
LIN {X 0,Y 446.418,Z 466.487,A -85,B 0,C 180,E1 -8796.823,E2 -8796.823} C_VEL
LIN {X 0,Y 446.433,Z 466.489,A -85,B 0,C 180,E1 -8799.737,E2 -8799.737} C_VEL
LIN {X 0,Y 446.453,Z 466.5,A -85,B 0,C 180,E1 -8802.597,E2 -8802.597} C_VEL
LIN {X 0,Y 446.461,Z 466.493,A -85,B 0,C 180,E1 -8805.412,E2 -8805.412} C_VEL
LIN {X 0,Y 446.535,Z 466.486,A -85,B 0,C 180,E1 -8808.194,E2 -8808.194} C_VEL
LIN {X 0,Y 446.589,Z 466.478,A -85,B 0,C 180,E1 -8811.858,E2 -8811.858} C_VEL
LIN {X 0,Y 446.639,Z 466.473,A -85,B 0,C 180,E1 -8814.583,E2 -8814.583} C_VEL
LIN {X 0,Y 446.7,Z 466.461,A -85,B 0,C 180,E1 -8817.295,E2 -8817.295} C_VEL
LIN {X 0,Y 446.783,Z 466.452,A -85,B 0,C 180,E1 -8820,E2 -8820} C_VEL
LIN {X 0,Y 446.699,Z 466.463,A -85,B 0,C 180,E1 -8822.705,E2 -8822.705} C_VEL
LIN {X 0,Y 446.636,Z 466.476,A -85,B 0,C 180,E1 -8826.324,E2 -8826.324} C_VEL
